VAR
	m_Out:INT;
	m_in: LREAL;
END_VAR

IF Enable THEN
	IF ABS(MaxValue) > 0.0 THEN
		m_in:=LIMIT(0, In, Set_MaxValue);
		m_Out:=REAL_TO_INT(m_In /MaxValue*32767) + AnalogOffset;
		out:=LIMIT(0, m_out, 32767);
	ELSE
		out:=AnalogOffset;
	END_IF
ELSE
	out:=AnalogOffset;
END_IF

END_FUNCTION_BLOCK

// ---- POUs/002_Modbus/PRG_SerialComm.TcPOU
PROGRAM PRG_SerialComm
VAR
	CmdSendData1,CmdSendData2,CmdSendData3		: SendData; //将任何类型的变量的内容发送到与输入变量TxBuffer对应的接口。只要Busy=TRUE，传输就没有完成。当Busy=FALSE和Error=0时，数据已成功发送
	StsReceiveData1,StsReceiveData2	: ReceiveData;
	DataRecive1     :ARRAY[1..16]OF BYTE;	
	Prefix1 : ARRAY[1..5] OF BYTE :=[16#46,16#51,16#0C,16#32,16#02];
	
	Dely1,Dely2:Tc2_Standard.TON;
	clearbuf1,clearbuf2,clearbuf3,clearbuf4:Tc2_SerialCom.ClearComBuffer;
	i,j: INT;
	
	level:ARRAY[1..10] OF LREAL;	
	(*******************UV mode****************************)
	DataSend_uv_mode					:ARRAY[1..11]OF BYTE:=[16#01,16#10,16#00,16#C0,16#00,16#01,16#02,16#00,16#11,16#77,16#5C];//232
	DataRecive_uv_mode	    			:ARRAY[1..8] OF BYTE;
	DataRecive_uv_mode_correct			:ARRAY[1..8] OF BYTE:=[16#01,16#10,16#00,16#C0,16#00,16#01,16#01,16#F5];
	ton_Remote							:Tc2_Standard.TON;
	(*******************UV buad****************************)
	step_burd							:INT;
	DataSend_Buad_set					:ARRAY[1..17] OF BYTE;
	DataSend_Buad						:ARRAY[1..19] OF BYTE;
	DataRecive_Buad_correct				:ARRAY[1..8] OF BYTE:=[16#01,16#10,16#01,16#20,16#00,16#05,16#00,16#3C];
	DataRecive_Buad						:ARRAY[1..8] OF BYTE;
	EN_Buad:DINT;
	HMI_Buad:INT:=2;//1：9600,2:57600,3:115200
	CRC16_Send_Buad:WORD;
	(*******************UV power****************************)
	step_set_power							:INT;
	DataSend_Power_set						:ARRAY[1..41] OF BYTE;
	DataSend_Power						    :ARRAY[1..43] OF BYTE;
	DataReceive_Power						:ARRAY[1..8] OF BYTE;
	CRC16_Send_Power:WORD;
	UV_power_old_L							:DINT;//上一次能量
	UV_power_old_R							:DINT;//上一次能量
	UV_Power_r_trig:						Tc2_Standard.R_TRIG;//能量变化
	UV_Power_send_f_trig					:Tc2_Standard.F_TRIG;
	(*******************UV STATE****************************)
	step_read_state:INT;
	DataSend_State						:ARRAY[1..8] OF BYTE:=[16#01,16#03,16#00,16#CB,16#00,16#1A,16#B5,16#FF];
	DataRecive_State					:ARRAY[1..57] OF BYTE;
	Prefix_DataRecive_State: ARRAY[1..3] OF BYTE :=[16#01,16#03,16#34];
	
	(*******************UV version****************************)
	step_read_version	:INT;
	DataSend_Version	:ARRAY[1..8] OF BYTE:=[16#01,16#03,16#00,16#AE,16#00,16#10,16#25,16#E7];
	DataRecive_Version	:ARRAY[1..37] OF BYTE;
	Prefix_DataRecive_Version: ARRAY[1..3] OF BYTE :=[16#01,16#03,16#20];
	soft_version :ARRAY[0..2] OF WORD;
	soft_date    :ARRAY[0..2] OF WORD;//年，月，日
	hardware_version :ARRAY[0..2] OF WORD;
	hardware_date:ARRAY[0..2] OF WORD;//年，月，日
		
	(*******************UV first light****************************)
	step_first_light        :INT;
	DataSend_First_light	:ARRAY[1..8] OF BYTE:=[16#01,16#03,16#02,16#12,16#00,16#06,16#64,16#75];
	DataRecive_First_light	:ARRAY[1..17] OF BYTE;
	Prefix_DataRecive_First_light: ARRAY[1..3] OF BYTE :=[16#01,16#03,16#0C];
	
	(*******************UV Read the accumulated working time****************************)
	step_acc_working_time       :INT;
	DataSend_Acc_working_time 	:ARRAY[1..8] OF BYTE:=[16#01,16#03,16#00,16#E4,16#00,16#20,16#04,16#25];
	DataRecive_Acc_working_time	:ARRAY[1..69] OF BYTE;
	Prefix_DataRecive_Acc_working_time: ARRAY[1..3] OF BYTE :=[16#01,16#03,16#40];


	
	Receive_data_F_trig:Tc2_Standard.F_TRIG;
	
	TON_Timeout:ARRAY[1..4] OF Tc2_Standard.TON;

	
	Main_step_UV:INT;
	
	
		
	uv_power_left_t,uv_power_right_t:DINT;
	bHibyte,bLobyte:BYTE;
	
	error_count_test:ARRAY[1..10] OF DINT;
	error_trig_test:ARRAY[1..10] OF Tc2_Standard.R_TRIG;
	
	CMD_Burd,CMD_Read_Version,CMD_Read_First_light,CMD_Read_Acc_working_time:BOOL;
	
	ton_case:Tc2_Standard.TON;
	
END_VAR

(****************MainTankLevel***************)
COM1_MainTankLevel();

(*********************************UV**************************************)
(*********************clear buff******************				
Dely1(IN:=NOT Dely1.Q , PT:=T#500MS , Q=> , ET=> );	
IF Dely1.Q THEN 
		clearbuf3(Buffer:=TXBUFFER2  );
		clearbuf4(Buffer:=RXBUFFER2   );	
END_IF
*)
(*****************timeout,自复位***************************)
TON_Timeout[1](IN:= NOT StsReceiveData2.busy  , PT:=T#2S , Q=> , ET=> );
TON_Timeout[2](IN:=StsReceiveData2.busy  , PT:=T#2S , Q=> , ET=> );
IF TON_Timeout[1].Q OR TON_Timeout[2].Q THEN 
	GVL.UV_timeout:=TRUE;
ELSE
	GVL.UV_timeout:=FALSE;
END_IF


(*********************UV_pro*******************)
COM2_UVLed_Set_Power();

IF Axis[1].Ref.Status.NotMoving THEN 
	CASE Main_step_UV OF
	0:
		IF CMD_Burd THEN 
			Main_step_UV:=10;
		ELSIF CMD_Read_Version THEN 
			Main_step_UV:=20;
		ELSIF CMD_Read_First_light THEN 
			Main_step_UV:=30;
		ELSIF CMD_Read_Acc_working_time THEN 
			Main_step_UV:=40;
		ELSE 
			Main_step_UV:=50;
		END_IF
	10://COM2_UVLedburd 
		CMD_Burd:=FALSE;
		_10_COM2_UVLed_burd();
		ton_case(IN:=TRUE , PT:=T#1S , Q=> , ET=> );
		Receive_data_F_trig(CLK:=StsReceiveData2.busy , Q=> );
		IF ton_case.Q OR Receive_data_F_trig.Q  THEN 
			ton_case(IN:=FALSE);
			step_burd:=0;
			Main_step_UV:=0;
		END_IF
	20://CMD_Read_Version
		CMD_Read_Version:=FALSE;
		_20_COM2_UVLed_Version();
		ton_case(IN:=TRUE , PT:=T#1S , Q=> , ET=> );
		Receive_data_F_trig(CLK:=StsReceiveData2.busy , Q=> );
		IF ton_case.Q OR Receive_data_F_trig.Q THEN 
			ton_case(IN:=FALSE);
			step_read_version:=0;
			Main_step_UV:=0;
		END_IF
		
	30://CMD_Read_First_light
		CMD_Read_First_light:=FALSE;
		_30_COM2_UVLed_First_light();
		ton_case(IN:=TRUE , PT:=T#1S , Q=> , ET=> );
		Receive_data_F_trig(CLK:=StsReceiveData2.busy , Q=> );
		IF ton_case.Q THEN 
			ton_case(IN:=FALSE);
			step_first_light:=0;		
			Main_step_UV:=0;
		END_IF
	40://CMD_Read_Acc_working_time
		CMD_Read_Acc_working_time:=FALSE;
		_40_COM2_UVLed_Acc_working_time();
		ton_case(IN:=TRUE , PT:=T#1S , Q=> , ET=> );
		Receive_data_F_trig(CLK:=StsReceiveData2.busy , Q=> );
		IF ton_case.Q THEN 
			ton_case(IN:=FALSE);
			step_acc_working_time:=0;
			Main_step_UV:=0;
		END_IF
	50:		
		_50_COM2_UVLed_Read_State();
		IF CMD_Burd OR CMD_Read_Version OR CMD_Read_First_light OR CMD_Read_Acc_working_time THEN
			Main_step_UV:=0;
		END_IF 
	END_CASE

END_IF

ACTION _10_COM2_UVLed_burd:
IF HMI_Buad=1 THEN  //9600
		DataSend_Buad_set[8]:=16#00;
		DataSend_Buad_set[9]:=16#00;
		DataSend_Buad_set[10]:=16#25;
		DataSend_Buad_set[11]:=16#80;
	ELSIF HMI_Buad=2 THEN //57600
		DataSend_Buad_set[8]:=16#00;
		DataSend_Buad_set[9]:=16#00;
		DataSend_Buad_set[10]:=16#E1;
		DataSend_Buad_set[11]:=16#00;
	ELSIF HMI_Buad=3 THEN //115200
		DataSend_Buad_set[8]:=16#00;
		DataSend_Buad_set[9]:=16#01;
		DataSend_Buad_set[10]:=16#C2;
		DataSend_Buad_set[11]:=16#00;
	END_IF
	DataSend_Buad_set[1]:=16#01; DataSend_Buad_set[2]:=16#10;DataSend_Buad_set[3]:=16#01;
	DataSend_Buad_set[4]:=16#20; DataSend_Buad_set[5]:=16#00;DataSend_Buad_set[6]:=16#05;
	DataSend_Buad_set[7]:=16#0A; 
	DataSend_Buad_set[12]:=16#00; DataSend_Buad_set[13]:=16#00;//校验位
	DataSend_Buad_set[14]:=16#00;DataSend_Buad_set[15]:=16#08;//停止位
	DataSend_Buad_set[16]:=16#00;DataSend_Buad_set[17]:=16#01;//奇偶校验

	MEMCPY(destAddr:=ADR(DataSend_Buad) , srcAddr:=ADR(DataSend_Buad_set) , n:=SIZEOF(DataSend_Buad_set) );
	
	CRC16_Send_Buad:=MEM.CRC16_Modbus(pMemoryBlock:= ADR(DataSend_Buad_set) , uiLength:=SIZEOF(DataSend_Buad_set) );	
	DataSend_Buad[19]:=WORD_TO_BYTE(CRC16_Send_Buad/255);  // crc h
	DataSend_Buad[18]:=WORD_TO_BYTE(CRC16_Send_Buad);			//CRCL
CASE step_burd OF
0://
10://波特率设置	
	IF NOT  StsReceiveData2.busy THEN 
		CmdSendData2(
			pSendData:= ADR(DataSend_Buad), 
			Length:= 19, 
			Busy=> , 
			Error=> , 
			TXbuffer:= TXBUFFER2);
		step_burd:=20;
	END_IF
20://	接收，比较  波特率
		StsReceiveData2(
			pPrefix:= , 
			LenPrefix:=, 
			pSuffix:= , 
			LenSuffix:= , 
			pReceiveData:= ADR(DataRecive_Buad), 
			SizeReceiveData:= SIZEOF(DataRecive_Buad), 
			Timeout:=T#500MS , 
			Reset:= , 
			DataReceived=> , 
			busy=> , 
			Error=> , 
			RxTimeout=> , 
			LenReceiveData=> , 
			RXbuffer:= RXBUFFER2);
			
			EN_Buad:=MEMCMP(pBuf1:=ADR(DataRecive_Buad) , pBuf2:=ADR(DataRecive_Buad_correct) , n:=SIZEOF(DataRecive_Buad_correct) );
			
			//step_burd:=0;

			
END_CASE
(*
40://  接收，比较  模式
 	StsReceiveData2(
		pPrefix:= , 
		LenPrefix:=, 
		pSuffix:= , 
		LenSuffix:= , 
		pReceiveData:= ADR(DataRecive_uv_mode), 
		SizeReceiveData:= SIZEOF(DataRecive_uv_mode), 
		Timeout:=T#500MS , 
		Reset:= , 
		DataReceived=> , 
		busy=> , 
		Error=> , 
		RxTimeout=> , 
		LenReceiveData=> , 
		RXbuffer:= RXBUFFER2);
	
 	EN_mode:=MEMCMP(pBuf1:=ADR(DataRecive_uv_mode) , pBuf2:=ADR(DataRecive_uv_mode_correct) , n:=SIZEOF(DataRecive_uv_mode_correct) );
	step_UV:=0;
	(*IF EN_mode=0 THEN 
		step_UV:=0;
	ELSE 
		step_UV:=200;
	END_IF
	*)
*)
END_ACTION

ACTION _20_COM2_UVLed_Version:
CASE step_read_version OF 		
0:
	CmdSendData2(
				pSendData:= ADR(DataSend_Version), 
				Length:= 8, 
				Busy=> , 
				Error=> , 
				TXbuffer:= TXBUFFER2);
		step_read_version:=10;
10:		
		StsReceiveData2(
				pPrefix:=ADR(Prefix_DataRecive_Version) , 
				LenPrefix:=3, 
				pSuffix:= , 
				LenSuffix:= , 
				pReceiveData:= ADR(DataRecive_Version), 
				SizeReceiveData:= SIZEOF(DataRecive_Version), 
				Timeout:=T#500MS , 
				Reset:= , 
				DataReceived=> , 
				busy=> , 
				Error=> , 
				RxTimeout=> , 
				LenReceiveData=> , 
				RXbuffer:= RXBUFFER2);
		
		
20:
		;
END_CASE
END_ACTION

ACTION _30_COM2_UVLed_First_light:
CASE step_first_light OF 		
0:
	CmdSendData2(
				pSendData:= ADR(DataSend_First_light), 
				Length:= 8, 
				Busy=> , 
				Error=> , 
				TXbuffer:= TXBUFFER2);
		step_read_version:=10;
10:		
		StsReceiveData2(
				pPrefix:=ADR(Prefix_DataRecive_First_light) , 
				LenPrefix:=3, 
				pSuffix:= , 
				LenSuffix:= , 
				pReceiveData:= ADR(DataRecive_First_light), 
				SizeReceiveData:= SIZEOF(DataRecive_First_light), 
				Timeout:=T#500MS , 
				Reset:= , 
				DataReceived=> , 
				busy=> , 
				Error=> , 
				RxTimeout=> , 
				LenReceiveData=> , 
				RXbuffer:= RXBUFFER2);
		
20:
		;
END_CASE
END_ACTION

ACTION _40_COM2_UVLed_Acc_working_time:
CASE step_acc_working_time OF 		
0:
	CmdSendData2(
				pSendData:= ADR(DataSend_Acc_working_time), 
				Length:= 8, 
				Busy=> , 
				Error=> , 
				TXbuffer:= TXBUFFER2);
		step_read_version:=10;
10:		
		StsReceiveData2(
				pPrefix:=ADR(Prefix_DataRecive_Acc_working_time) , 
				LenPrefix:=3, 
				pSuffix:= , 
				LenSuffix:= , 
				pReceiveData:= ADR(DataRecive_Acc_working_time), 
				SizeReceiveData:= SIZEOF(DataRecive_Acc_working_time), 
				Timeout:=T#500MS , 
				Reset:= , 
				DataReceived=> , 
				busy=> , 
				Error=> , 
				RxTimeout=> , 
				LenReceiveData=> , 
				RXbuffer:= RXBUFFER2);
		
20:
		;
END_CASE
END_ACTION

ACTION _50_COM2_UVLed_Read_State:
(**************读取灯的能量和温度**************************************************)
GVL.HMI_TEMP_L:=BYTE_TO_INT(DataRecive_State[7]);
GVL.HMI_TEMP_R:=BYTE_TO_INT(DataRecive_State[11]);
GVL.HMI_power_L:=BYTE_TO_INT(DataRecive_State[5]);
GVL.HMI_power_R:=BYTE_TO_INT(DataRecive_State[9]);

(******************************************main*****************************************
		StsReceiveData2(
				pPrefix:=ADR(Prefix_DataRecive_State) , 
				LenPrefix:=3, 
				pSuffix:= , 
				LenSuffix:= , 
				pReceiveData:= ADR(DataRecive_State), 
				SizeReceiveData:= SIZEOF(DataRecive_State), 
				Timeout:=T#500MS , 
				Reset:= , 
				DataReceived=> , 
				busy=> , 
				Error=> , 
				RxTimeout=> , 
				LenReceiveData=> , 
				RXbuffer:= RXBUFFER2);
		*)
CASE step_read_state  OF
	
0://读状态，发送
	Dely2(IN:=NOT Dely2.Q  , PT:=T#1000MS , Q=> , ET=> );	
	IF Dely2.Q  THEN 
		
		CmdSendData2(
				pSendData:= ADR(DataSend_State), 
				Length:= 8, 
				Busy=> , 
				Error=> , 
				TXbuffer:= TXBUFFER2);
		step_read_state:=10;    
	END_IF     
10://接收
	Dely2(IN:=false);
	StsReceiveData2(
				pPrefix:=ADR(Prefix_DataRecive_State) , 
				LenPrefix:=3, 
				pSuffix:= , 
				LenSuffix:= , 
				pReceiveData:= ADR(DataRecive_State), 
				SizeReceiveData:= SIZEOF(DataRecive_State), 
				Timeout:=T#500MS , 
				Reset:= , 
				DataReceived=> , 
				busy=> , 
				Error=> , 
				RxTimeout=> , 
				LenReceiveData=> , 
				RXbuffer:= RXBUFFER2);
		step_read_state:=20;  
20://处理数据	 	
		IF DataRecive_State[7]=16#FF THEN //温度异常
				GVL.UV_error_L:=TRUE;
				step_read_state:=100;
		ELSIF  DataRecive_State[11]=16#FF THEN //温度异常
				GVL.UV_error_R:=TRUE;
				step_read_state:=100;	
		ELSIF	DataRecive_State[13]<>16#11	THEN 	//不是232控制
				step_read_state:=30;
		ELSIF  	DataRecive_State[13]=16#11 AND DataRecive_State[7]<>16#FF AND 
			DataRecive_State[11]<>16#FF AND NOT  GVL.UV_error_L  AND NOT GVL.UV_error_R THEN 
				step_read_state:=0;		
		END_IF
		//step_read_state:=0;
30://设定模式RS232		
	   CmdSendData2(
			pSendData:= ADR(DataSend_uv_mode), 
			Length:= 11, 
			Busy=> , 
			Error=> , 
			TXbuffer:= TXBUFFER2);	
   		step_read_state:=0;
					
100://error
			IF GVL_API.stUVLed[1].SetOff OR  GVL_API.stUVLed[2].SetOff THEN 
				GVL.UV_error_L:=FALSE;
				GVL.UV_error_R:=FALSE;
				step_read_state:=0;
			END_IF				
END_CASE
(**************remote***********************)
ton_Remote(IN:=DataRecive_State[13]<>16#11 , PT:=T#5S , Q=> , ET=> );
IF DataRecive_State[13]=16#11 THEN 
	GVL.UVisRemote:=TRUE;
ELSIF ton_Remote.Q THEN 
	GVL.UVisRemote:=FALSE;
END_IF
END_ACTION

ACTION COM1_MainTankLevel:
(************************通讯参数设置*******************)
//Dely1(IN:=TRUE , PT:=T#100MS , Q=> , ET=> );

StsReceiveData1(
	pPrefix:=ADR(Prefix1) , 
	LenPrefix:=5 , 
	pSuffix:= , 
	LenSuffix:= , 
	pReceiveData:= ADR(DataRecive1), 
	SizeReceiveData:= SIZEOF(DataRecive1), 
	Timeout:=T#500MS , 
	Reset:= , 
	DataReceived=> , 
	busy=> , 
	Error=> , 
	RxTimeout=> , 
	LenReceiveData=> , 
	RXbuffer:= RXBUFFER1);

(****************计算********************)
FOR i:=6 TO 15 DO 
	IF DataRecive1[i]<>255 AND DataRecive1[i]<=10 THEN 
		level[i-5]:=BYTE_TO_LREAL(DataRecive1[i]);
	ELSE
		level[i-5]:=0;
	END_IF
END_FOR
GVL.MainTankLevel[1]:=level[5];//LC
GVL.MainTankLevel[2]:=level[6];//LM
GVL.MainTankLevel[3]:=level[4];//Y
GVL.MainTankLevel[4]:=level[3];//M
GVL.MainTankLevel[5]:=level[2];//C
GVL.MainTankLevel[6]:=level[1];//K
GVL.MainTankLevel[7]:=level[7];//W
GVL.MainTankLevel[8]:=level[8];//P
GVL.MainTankLevel[9]:=level[9];//FU
GVL.MainTankLevel[10]:=level[10];//WAST

(*****************timeout,自复位***************************)
TON_Timeout[3](IN:= NOT StsReceiveData1.busy  , PT:=T#2S , Q=> , ET=> );
TON_Timeout[4](IN:=StsReceiveData1.busy  , PT:=T#2S , Q=> , ET=> );
IF TON_Timeout[3].Q OR TON_Timeout[4].Q THEN 
	gvl.MainTankLevel_timeout:=TRUE;
ELSE
	gvl.MainTankLevel_timeout:=FALSE;
END_IF
END_ACTION

ACTION COM2_UVLed_1:
GVL.HMI_TEMP_L:=BYTE_TO_INT(DataRecive_State[7]);
GVL.HMI_TEMP_R:=BYTE_TO_INT(DataRecive_State[11]);
GVL.HMI_power_L:=BYTE_TO_INT(DataRecive_State[5]);
GVL.HMI_power_R:=BYTE_TO_INT(DataRecive_State[9]);
(******************************************UV******************************************)
Dely2(IN:=NOT Dely2.Q  , PT:=T#100MS , Q=> , ET=> );	
IF Dely2.Q AND NOT UV_Power_r_trig.Q THEN 
		CmdSendData2(
				pSendData:= ADR(DataSend_State), 
				Length:= 8, 
				Busy=> , 
				Error=> , 
				TXbuffer:= TXBUFFER2);	
		
END_IF
		StsReceiveData2(
				pPrefix:=ADR(Prefix_DataRecive_State) , 
				LenPrefix:=3, 
				pSuffix:= , 
				LenSuffix:= , 
				pReceiveData:= ADR(DataRecive_State), 
				SizeReceiveData:= SIZEOF(DataRecive_State), 
				Timeout:=T#500MS , 
				Reset:= , 
				DataReceived=> , 
				busy=> , 
				Error=> , 
				RxTimeout=> , 
				LenReceiveData=> , 
				RXbuffer:= RXBUFFER2);
				
(******************************************clear buff******************************************)				
Dely1(IN:=NOT Dely1.Q , PT:=T#500MS , Q=> , ET=> );	
IF Dely1.Q THEN 
		clearbuf3(Buffer:=TXBUFFER2  );
		clearbuf4(Buffer:=RXBUFFER2   );	
END_IF

(******************************************main******************************************)
CASE step_read_state  OF		
0://处理数据
		IF DataRecive_State[7]=16#FF THEN //温度异常
				GVL.UV_error_L:=TRUE;
				step_read_state:=50;
		ELSIF  DataRecive_State[11]=16#FF THEN //温度异常
				GVL.UV_error_R:=TRUE;
				step_read_state:=50;	
		ELSIF	DataRecive_State[13]<>16#11	THEN 	//不是232控制
				step_read_state:=30;
		ELSIF  	DataRecive_State[13]=16#11 AND DataRecive_State[7]<>16#FF AND 
			DataRecive_State[11]<>16#FF AND NOT  GVL.UV_error_L  AND NOT GVL.UV_error_R THEN 
				step_read_state:=50;		//状态正常，设置能量
		END_IF

30://设定模式RS232		
	   CmdSendData2(
			pSendData:= ADR(DataSend_uv_mode), 
			Length:= 11, 
			Busy=> , 
			Error=> , 
			TXbuffer:= TXBUFFER2);	
   		step_read_state:=0;


50:	//	设置能量
		IF NOT GVL.UV_error_L AND NOT  GVL.UV_error_R THEN 
			DataSend_Power_set[8]:=16#00;DataSend_Power_set[9]:=16#11;	//命令
		ELSE
			DataSend_Power_set[8]:=16#00;DataSend_Power_set[9]:=16#00;	//命令	停机
		END_IF
		
		DataSend_Power_set[1]:=16#01;DataSend_Power_set[2]:=16#10;
		DataSend_Power_set[3]:=16#01;DataSend_Power_set[4]:=16#A0;
		DataSend_Power_set[5]:=16#00;DataSend_Power_set[6]:=16#11;
		DataSend_Power_set[7]:=16#22;
		
		
		DataSend_Power_set[10]:=16#00;
		DataSend_Power_set[11]:=DINT_TO_BYTE(GVL.set_uv_power_left);//灯0能量100
		///DataSend_Power_set[11]:=DINT_TO_BYTE(uv_power_left_t);//灯0能量100
		DataSend_Power_set[12]:=16#00;DataSend_Power_set[13]:=GVL.set_uv_parts_left;//灯0段数最大6
		
		DataSend_Power_set[14]:=16#00;
		DataSend_Power_set[15]:=DINT_TO_BYTE(GVL.set_uv_power_right);//灯1能量100
		//DataSend_Power_set[15]:=DINT_TO_BYTE(uv_power_right_t);//灯1能量100
		DataSend_Power_set[16]:=16#00;DataSend_Power_set[17]:=GVL.set_uv_parts_right;//灯1段数最大6
		FOR j:=18 TO 41 DO 
			DataSend_Power_set[J]:=16#00;
		END_FOR
		
		MEMCPY(destAddr:=ADR(DataSend_Power) , srcAddr:=ADR(DataSend_Power_set) , n:=SIZEOF(DataSend_Power_set) );
		CRC16_Send_Power:=MEM.CRC16_Modbus(pMemoryBlock:= ADR(DataSend_Power_set) , uiLength:=SIZEOF(DataSend_Power_set) );
		DataSend_Power[43]:=WORD_TO_BYTE(CRC16_Send_Power/256);  // crc h
		DataSend_Power[42]:=WORD_TO_BYTE(CRC16_Send_Power);			//CRCL
		//bHibyte:=MEM.HighByte(wValue:=CRC16_Send_Power );
		//bLobyte:=MEM.LowByte(wValue:=CRC16_Send_Power );
		
	(*****************检测能量设置变化****************************)	
	UV_Power_r_trig(CLK:=UV_power_old_L<>GVL.set_uv_power_left OR UV_power_old_R<> GVL.set_uv_power_right , Q=> );
		//IF GVL.UV_error_L OR   GVL.UV_error_R OR UV_Power_r_trig.Q THEN 
			UV_power_old_L:=GVL.set_uv_power_left;
			UV_power_old_R:=GVL.set_uv_power_right;
			
			
	
		//END_IF
		
		IF NOT GVL.UV_error_L AND NOT  GVL.UV_error_R THEN 
			step_read_state:=0;
		ELSE
			step_read_state:=100;	//命令	停机
		END_IF
							
100://error
			IF GVL_API.stUVLed[1].SetOff OR  GVL_API.stUVLed[2].SetOff THEN 
				GVL.UV_error_L:=FALSE;
				GVL.UV_error_R:=FALSE;
				step_read_state:=0;
			END_IF			
END_CASE

			CmdSendData3(
					pSendData:= ADR(DataSend_Power), 
					Length:= SIZEOF(DataSend_Power), 
					Busy=> , 
					Error=> , 
					TXbuffer:= TXBUFFER2);	


	 
	 
(*****************timeout,自复位***************************)
TON_Timeout[1](IN:= NOT StsReceiveData2.busy  , PT:=T#2S , Q=> , ET=> );
TON_Timeout[2](IN:=StsReceiveData2.busy  , PT:=T#2S , Q=> , ET=> );
IF TON_Timeout[1].Q OR TON_Timeout[2].Q THEN 
	GVL.UV_timeout:=TRUE;
ELSE
	GVL.UV_timeout:=FALSE;
END_IF
END_ACTION

ACTION COM2_UVLed_Set_Power:
//设置能量
		IF NOT GVL.UV_error_L AND NOT  GVL.UV_error_R THEN 
			DataSend_Power_set[8]:=16#00;DataSend_Power_set[9]:=16#11;	//命令
		ELSE
			DataSend_Power_set[8]:=16#00;DataSend_Power_set[9]:=16#00;	//命令	停机
		END_IF
		
		DataSend_Power_set[1]:=16#01;DataSend_Power_set[2]:=16#10;
		DataSend_Power_set[3]:=16#01;DataSend_Power_set[4]:=16#A0;
		DataSend_Power_set[5]:=16#00;DataSend_Power_set[6]:=16#11;
		DataSend_Power_set[7]:=16#22;
		
		
		DataSend_Power_set[10]:=16#00;
		
		DataSend_Power_set[11]:=DINT_TO_BYTE(GVL.set_uv_power_left);//灯0能量100
		//DataSend_Power_set[11]:=DINT_TO_BYTE(uv_power_left_t);//灯0能量100
		
		DataSend_Power_set[12]:=16#00;DataSend_Power_set[13]:=GVL.set_uv_parts_left;//灯0段数最大6
		
		DataSend_Power_set[14]:=16#00;
		
		DataSend_Power_set[15]:=DINT_TO_BYTE(GVL.set_uv_power_right);//灯1能量100
		//DataSend_Power_set[15]:=DINT_TO_BYTE(uv_power_right_t);//灯1能量100
		
		DataSend_Power_set[16]:=16#00;DataSend_Power_set[17]:=GVL.set_uv_parts_right;//灯1段数最大6
		FOR j:=18 TO 41 DO 
			DataSend_Power_set[J]:=16#00;
		END_FOR
		
		MEMCPY(destAddr:=ADR(DataSend_Power) , srcAddr:=ADR(DataSend_Power_set) , n:=SIZEOF(DataSend_Power_set) );
		CRC16_Send_Power:=MEM.CRC16_Modbus(pMemoryBlock:= ADR(DataSend_Power_set) , uiLength:=SIZEOF(DataSend_Power_set) );
		//DataSend_Power[43]:=WORD_TO_BYTE(CRC16_Send_Power/256);  // crc h
		//DataSend_Power[42]:=WORD_TO_BYTE(CRC16_Send_Power);			//CRCL
		DataSend_Power[43]:=MEM.HighByte(wValue:=CRC16_Send_Power);
		DataSend_Power[42]:=MEM.LowByte(wValue:=CRC16_Send_Power);

CmdSendData3(
			pSendData:= ADR(DataSend_Power), 
			Length:= SIZEOF(DataSend_Power), 
			Busy=> , 
			Error=> , 
			TXbuffer:= TXBUFFER2);
	UV_Power_send_f_trig(CLK:=CmdSendData3.Busy , Q=> );
(*
CASE step_set_power OF
0:
(*****************检测能量设置变化****************************)
UV_Power_r_trig(CLK:=UV_power_old_L<>GVL.set_uv_power_left OR UV_power_old_R<> GVL.set_uv_power_right , Q=> );
	IF UV_Power_r_trig.Q THEN 
			UV_power_old_L:=GVL.set_uv_power_left;
			UV_power_old_R:=GVL.set_uv_power_right;
		step_set_power:=10;
	END_IF
10:
	CmdSendData3(
			pSendData:= ADR(DataSend_Power), 
			Length:= SIZEOF(DataSend_Power), 
			Busy=> , 
			Error=> , 
			TXbuffer:= TXBUFFER2);
	UV_Power_send_f_trig(CLK:=CmdSendData3.Busy , Q=> );
	//IF UV_Power_send_f_trig.Q AND CmdSendData3.Error=0 THEN 
			step_set_power:=0;
	//END_IF
END_CASE
*)
END_ACTION

END_PROGRAM

// ---- POUs/002_Modbus/P_Modbus_RTU.TcPOU
PROGRAM P_Modbus_RTU
VAR
	(*********************RTU******************************)
	master:ARRAY[1..2] OF    ModbusRtuMaster_KL6x22B;
    start:ARRAY[1..2] OF  BOOL:=[TRUE];
	step:ARRAY[1..2] OF  INT;
	
	com1_station:ARRAY[1..5] OF stRtu;
	
	tab_vac_measure	:ARRAY[1..2] OF WORD;//负压表值
	tab_vac_set		:ARRAY[1..2] OF WORD;//负压表值
	sub_pressure_measure	: LREAL;//sub测量正压
	sub_pressure_set		: LREAL;//sun正压设定值
	sub_vac_c_measure		: LREAL;//sub彩色负压值
	sub_vac_w_measure		: LREAL;//sub白色负压值
	sub_vac_c_set			: LREAL;//sub彩色负压设定值
	sub_vac_w_set			: LREAL;//sub白色负压设定值
	
	cycle_time:INT;
	count_time:INT:=5;
	i,j:INT;	
	error_trig :ARRAY[1..10] OF Tc2_Standard.R_TRIG;
	error_count:ARRAY[1..10] OF DINT;//错误计数
	station_error_trig:ARRAY[1..10] OF Tc2_Standard.R_TRIG;	
	station_error AT%Q*:ARRAY[1..10] OF BOOL;
	test_send:BOOL;
END_VAR

VAR PERSISTENT
	break_systime:ARRAY[1..10] OF DATE_AND_TIME;
END_VAR

ACT();

(******************************************台面负压****************************************************)
	(*原本接收10代表1KPA，但修改温控表，使10代表1*)
	(**********READ****负数=正数按位取反+1******************************)
	IF com1_station[1]._04readarray[1].15=0 THEN 
		GVL_API.stTableVacuum[1].vacuum_measured:=WORD_TO_LREAL(com1_station[1]._04readarray[1])/100;
	ELSE 
		GVL_API.stTableVacuum[1].vacuum_measured:=WORD_TO_LREAL(NOT(com1_station[1]._04readarray[1]-1))/100;
	END_IF
	(***************台面负压****write****)	
	com1_station[1]._06writesinglearray[1]:=NOT (LREAL_TO_WORD(GVL_API.stTableVacuum[1].setpoint*100))+1;///负数，反吗+1
	(***************台面负压****writPID*)
	IF 	GVL_API.stTableVacuum[1].ctrlP >0 THEN 	//P 不能为0
		com1_station[1]._06writesinglearray_PID[2]:=LREAL_TO_WORD(GVL_API.stTableVacuum[1].ctrlP*10);//制冷端P
	ELSE 
		com1_station[1]._06writesinglearray_PID[2]:=LREAL_TO_WORD(10*10);//制冷端P
	END_IF
		com1_station[1]._06writesinglearray_PID[4]:=LREAL_TO_WORD(GVL_API.stTableVacuum[1].ctrlI);
		com1_station[1]._06writesinglearray_PID[6]:=LREAL_TO_WORD(GVL_API.stTableVacuum[1].ctrlD);
	
		
(***************温湿度****************)
		gvl.humidity_measured:=	WORD_TO_LREAL(com1_station[3]._03readarray[1])/10;
		IF com1_station[3]._03readarray[1].15=0 THEN 
			gvl.temp_measured:=WORD_TO_LREAL(com1_station[3]._03readarray[2])/10;
		ELSIF com1_station[3]._03readarray[1].15=1 THEN
			gvl.temp_measured:= WORD_TO_LREAL(NOT(com1_station[3]._03readarray[2]-1))/10;
		END_IF
		
		
		
(**************二级墨盒正负压****************
	(**********SUB VAC 正压**************)
	sub_pressure_measure:=  WORD_TO_LREAL( com1_station[4]._03readarray[1])/1000;   //当前值
	
	com1_station[4]._03writearray[1]:=LREAL_TO_WORD(sub_pressure_set*1000);//正压设定
	com1_station[4]._03writearray[4]:=1;//正压自启动
	com1_station[4]._03writearray[4]:=12;//正压电机速度
	
	(**********SUB VAC 负压**************)
	sub_vac_c_measure:=WORD_TO_LREAL(com1_station[5]._03readarray[1])/1000;
	sub_vac_w_measure:=WORD_TO_LREAL(com1_station[5]._03readarray[2])/1000;
	
	com1_station[5]._03writearray[1]:=LREAL_TO_WORD(sub_vac_c_set*1000);
	com1_station[5]._03writearray[2]:=LREAL_TO_WORD(sub_vac_w_set*1000);
	com1_station[5]._03writearray[3]:=3;
	com1_station[5]._03writearray[4]:=3;
*)

ACTION ACT:
CASE step[1] OF 
0: //初始状态
		IF start[1] THEN
			step[1]:=10;
			cycle_time:=0;
		END_IF	
10://站1 04口读操作  真空吸附			
			IF cycle_time>=count_time THEN 
				cycle_time:=0;	
				FOR j:=1 TO 10 DO 
					error_count[j]:=0;
				END_FOR		
			END_IF
						
			master[1].ReadInputRegs(
				UnitID:= 1, 
				Quantity:=4, 
				MBAddr:= 16#03E8, 
				cbLength:= SIZEOF(com1_station[1]._04readarray), 
				pMemoryAddr:= ADR(com1_station[1]._04readarray), 
				Execute:= TRUE, 
				Timeout:= T#200MS);	
											
				IF NOT master[1].BUSY  THEN
					master[1].ReadRegs(Execute:= FALSE, );
					cycle_time:=cycle_time+1;
					step[1]:=20;									
				END_IF
				
				station_error_trig[1](CLK:=master[1].error , Q=> );	
				IF station_error_trig[1].Q THEN 
					error_count[1]:=error_count[1]+1;
				END_IF
20://站1 06口写操作	,设定负压	
			master[1].WriteSingleRegister(
				UnitID:= 1, 
				Quantity:=1, 
				MBAddr:= 0, 
				cbLength:= 2, 
				pMemoryAddr:= ADR(com1_station[1]._06writesinglearray[1]), 
				Execute:= TRUE, 
				Timeout:= T#200MS, 
				BUSY=> , 
				Error=> , 
				ErrorId=> , 
				cbRead=> );			
						
				IF NOT master[1].BUSY  THEN
					master[1].ReadRegs(Execute:= FALSE, );
					step[1]:=21;									
				END_IF
				
				station_error_trig[1](CLK:=master[1].error , Q=> );	
				IF station_error_trig[1].Q THEN 
					error_count[1]:=error_count[1]+1;
				END_IF
21://站1 06口写操作	,设定PID
			master[1].WriteRegs(
				UnitID:= 1, 
				Quantity:=SIZEOF(com1_station[1]._06writesinglearray_PID)/2, 
				MBAddr:= 16#0065, 
				cbLength:= SIZEOF(com1_station[1]._06writesinglearray_PID), 
				pMemoryAddr:= ADR(com1_station[1]._06writesinglearray_PID), 
				Execute:= TRUE, 
				Timeout:= T#200MS, 
				BUSY=> , 
				Error=> , 
				ErrorId=> , 
				cbRead=> );	
				
				
				station_error_trig[1](CLK:=master[1].error , Q=> );	
				IF station_error_trig[1].Q THEN 
					error_count[1]:=error_count[1]+1;
				END_IF	
				IF cycle_time=count_time AND error_count[1]>=2 THEN 
					station_error[1]:=TRUE;
				END_IF

				IF NOT master[1].BUSY  THEN
					master[1].ReadRegs(Execute:= FALSE );
					step[1]:=50;											              		
				END_IF	
(*3://站2 04口读操作
			master[1].ReadInputRegs(
				UnitID:= 2, 
				Quantity:=4, 
				MBAddr:= 16#03E8, 
				cbLength:= SIZEOF(com1_station[2]._04readarray), 
				pMemoryAddr:= ADR(com1_station[2]._04readarray), 
				Execute:= TRUE, 
				Timeout:= T#200MS, 
				 );	
					          
				station_error_trig[2](CLK:=master[1].error , Q=> );	
				IF station_error_trig[2].Q THEN 
					error_count_test[2]:=error_count_test[2]+1;
				END_IF	 
				IF cycle_time=count_time AND error_count_test[2]>=2 THEN 
					station_error[2]:=TRUE;
				END_IF

	
				IF NOT master[1].BUSY  THEN
					master[1].ReadRegs(Execute:= FALSE, );
					IF NOT station_error[2] THEN 
						step[1]:=4;									
					ELSIF station_error[2] THEN 
						step[1]:=5;	
					END_IF		              		
				END_IF					 	
4://站2 06口写操作			
			master[1].WriteSingleRegister(
				UnitID:= 2, 
				Quantity:=1, 
				MBAddr:= 0, 
				cbLength:= SIZEOF(com1_station[2]._06writesinglearray[1]), 
				pMemoryAddr:= ADR(com1_station[2]._06writesinglearray[1]), 
				Execute:= TRUE, 
				Timeout:= T#200MS, 
				BUSY=> , 
				Error=> , 
				ErrorId=> , 
				cbRead=> );			
				
			
				station_error_trig[2](CLK:=master[1].error , Q=> );	
				IF station_error_trig[2].Q THEN 
					error_count_test[2]:=error_count_test[2]+1;
				END_IF	
				IF cycle_time=count_time AND error_count_test[2]>=2 THEN 
					station_error[2]:=TRUE;
				END_IF

				IF NOT master[1].BUSY  THEN
					master[1].ReadRegs(Execute:= FALSE, );					
					IF NOT station_error[2] THEN 
						step[1]:=5;									
					ELSIF station_error[2] THEN 
						step[1]:=5;	
					END_IF		              		
				END_IF		
*)				 	
50://站3温湿度 03读
			master[1].ReadRegs(
				UnitID:= 3, 
				Quantity:=2, 
				MBAddr:= 0, 
				cbLength:= SIZEOF(com1_station[3]._03readarray), 
				pMemoryAddr:= ADR(com1_station[3]._03readarray), 
				Execute:= TRUE, 
				Timeout:= T#200MS, 
				 );	
							     
				station_error_trig[3](CLK:=master[1].error , Q=> );	
				IF station_error_trig[3].Q THEN 
					error_count[3]:=error_count[3]+1;
				END_IF
				IF cycle_time=count_time AND error_count[3]>=2 THEN 
					station_error[3]:=TRUE;
				END_IF
								
				IF NOT master[1].BUSY  THEN
					master[1].ReadRegs(Execute:= FALSE, );										
					step[1]:=10;															              		
				END_IF
				
(*							
6://站4，正压板 03口读操作  当前压墨板正压传感器值，单位0.1kPa	
	     master[1].ReadRegs(
				UnitID:= 16#48, 
				Quantity:=7, 
				MBAddr:= 0, 
				cbLength:= SIZEOF(com1_station[4]._03readarray), 
				pMemoryAddr:= ADR(com1_station[4]._03readarray), 
				Execute:= TRUE, 
				Timeout:= T#200MS, 
				 );	
							
				station_error_trig[4](CLK:=master[1].error , Q=> );	
				IF station_error_trig[4].Q THEN 
					error_count_test[4]:=error_count_test[4]+1;
				END_IF		
			
				IF cycle_time=count_time AND error_count_test[4]>=2 THEN 
					station_error[4]:=TRUE;
				END_IF
				
				IF NOT master[1].BUSY  THEN
					master[1].ReadRegs(Execute:= FALSE, );					
					IF NOT station_error[4] THEN 
						step[1]:=7;									
					ELSIF station_error[4] THEN 
						step[1]:=8;	
					END_IF		              		
				END_IF						     					
7://站4，正压板 03口写操作 设定的压墨值，单位0.1kPa，绝对值。
		master[1].WriteRegs(
				UnitID:= 16#48, 
				Quantity:=6, 
				MBAddr:= 1, 
				cbLength:= SIZEOF(com1_station[4]._03writearray), 
				pMemoryAddr:= ADR(com1_station[4]._03writearray), 
				Execute:= TRUE, 
				Timeout:= T#200MS, 
				BUSY=> , 
				Error=> , 
				ErrorId=> , 
				cbRead=> );			
						
				station_error_trig[4](CLK:=master[1].error , Q=> );	
				IF station_error_trig[4].Q THEN 
					error_count_test[4]:=error_count_test[4]+1;
				END_IF	
				IF cycle_time=count_time AND error_count_test[4]>=2 THEN 
					station_error[4]:=TRUE;
				END_IF
				
				IF NOT master[1].BUSY  AND NOT station_error[4]THEN
					master[1].ReadRegs(Execute:= FALSE, );	
					step[1]:=8;
				ELSIF station_error[4] THEN 
					step[1]:=8;
				END_IF
				IF NOT master[1].BUSY  THEN
					master[1].ReadRegs(Execute:= FALSE, );					
					IF NOT station_error[4] THEN 
						step[1]:=8;									
					ELSIF station_error[4] THEN 
						step[1]:=8;	
					END_IF		              		
				END_IF					     				
8://zhan 5负压板 03口读操作
		master[1].ReadRegs(
				UnitID:= 16#1D, 
				Quantity:=8, 
				MBAddr:= 0, 
				cbLength:= SIZEOF(com1_station[5]._03readarray), 
				pMemoryAddr:= ADR(com1_station[5]._03readarray), 
				Execute:= TRUE, 
				Timeout:= T#200MS, 
				 );	
				
				station_error_trig[5](CLK:=master[1].error , Q=> );	
				IF station_error_trig[5].Q THEN 
					error_count_test[5]:=error_count_test[5]+1;
				END_IF	

				IF cycle_time=count_time AND error_count_test[5]>=2 THEN 
					station_error[5]:=TRUE;
				END_IF
				
				IF NOT master[1].BUSY  THEN
					master[1].ReadRegs(Execute:= FALSE, );					
					IF NOT station_error[5] THEN 
						step[1]:=9;									
					ELSIF station_error[5] THEN 
						step[1]:=1;	
					END_IF		              		
				END_IF							     
9://zhan 5,负压板 03口写	
		master[1].WriteRegs(
				UnitID:= 16#1D, 
				Quantity:=4, 
				MBAddr:= 2, 
				cbLength:= SIZEOF(com1_station[5]._03writearray), 
				pMemoryAddr:= ADR(com1_station[5]._03writearray), 
				Execute:= TRUE, 
				Timeout:= T#200MS, 
				BUSY=> , 
				Error=> , 
				ErrorId=> , 
				cbRead=> );			
				
		
				station_error_trig[5](CLK:=master[1].error , Q=> );	
				IF station_error_trig[5].Q THEN 
					error_count_test[5]:=error_count_test[5]+1;
				END_IF	
				
				IF cycle_time=count_time AND error_count_test[5]>=2 THEN 
					station_error[5]:=TRUE;
				END_IF
					
				IF NOT master[1].BUSY  THEN
					master[1].ReadRegs(Execute:= FALSE, );					
					IF NOT station_error[5] THEN 
						step[1]:=1;									
					ELSIF station_error[5] THEN 
						step[1]:=1;	
					END_IF		              		
				END_IF	
*)
END_CASE

IF GVL_API.stTableVacuum[1].Setoff (*OR GVL_API.stTableVacuum[2].Setoff*) THEN 
	station_error[1]:=FALSE;
	//station_error[2]:=FALSE;
END_IF
IF   GVL_API.stSystemEnvironment.Reset THEN 
	station_error[3]:=FALSE;
END_IF


FOR i:=1 TO 5 DO
 error_trig[i](CLK:=station_error[i] , Q=> );
	IF  error_trig[i].Q THEN 
		break_systime[i]:=systime.dttime;		
	END_IF
END_FOR
END_ACTION

END_PROGRAM

// ---- POUs/003_Input_Output/P_API_IO.TcPOU
PROGRAM P_API_IO
VAR
END_VAR

gvl_api.stAxis[FastScan].Origin:=Axis[FastScan].IO.snHome;
gvl_api.stAxis[FastScan].LimitP:=Axis[FastScan].IO.snLimitP;
gvl_api.stAxis[Z_Axis].Origin:=Axis[Z_Axis].IO.snHome;
gvl_api.stAxis[Z_Axis].LimitP:=Axis[Z_Axis].IO.snLimitP;

END_PROGRAM

// ---- POUs/010_Motion/MotionBase/FB_Home_Z.TcPOU
FUNCTION_BLOCK FB_Home_Z
(*========================================
Execute需一直有效，功能块才会一直执行
先回原点，然后直接到等待位
==========================================*)
VAR_IN_OUT
	Axis				:AXIS_REF;	(* B *)
END_VAR
VAR_INPUT
	Execute				:BOOL;	(* B *)
	PosLimit			:BOOL;			(*正极限位信号*)
	NegLimit			:BOOL;			(*负极限位信号*)
	Position			:LREAL			(* B *) := DEFAULT_HOME_POSITION;
	HomeingVelo			:LREAL:=5;
	Standby_position	:LREAL;		//最终待机位
	bCalibrationCam 	:BOOL;	(* V *)	(* Beckhoff proprietary input *)
	rel_dis         	:LREAL:=10;  //碰到原点后，正向移动距离，在开始寻原点
	TimeOutSet       	:LREAL;//s
	reset				:BOOL;
	maxDistance:LREAL;
END_VAR
VAR_OUTPUT
	Done				:BOOL;	(* B *)
	Busy				:BOOL;	(* E *)
	Active				:BOOL;	(* E *)
	CommandAborted		:BOOL;	(* E *)
	Error				:BOOL;	(* B *)
	ErrorID				:UDINT;	(* E *)
	TimeOut				:BOOL;//回零超时
	HomeErr				:BOOL;//超过最大行程

END_VAR
VAR
	mcJog			:MC_Jog;
	mcHome			:MC_Home;
	mcRel           :MC_MoveRelative;
	mcAbs           :MC_MoveAbsolute;	
	mcStop			:MC_Stop;
	HomeStep		:INT;
	ton				:TON;
	StopDo			:BOOL;
	start_pos		:LREAL;
	start_r_trig:Tc2_Standard.R_TRIG;
END_VAR

ton(IN:=Execute , PT:=LREAL_TO_TIME(TimeOutSet*1000) , Q=> , ET=> );
IF ton.Q THEN 
	TimeOut:=TRUE;
	HomeStep	:=100;
END_IF

start_r_trig(CLK:=Execute , Q=> );
IF start_r_trig.Q THEN 
	start_pos:=Axis.NcToPlc.ActPos;
END_IF


IF  NOT Execute THEN
	mcJog.JogForward		:=FALSE;
	mcJog.JogBackwards		:=FALSE;
	mcHome.Execute			:=FALSE;
	mcRel.Execute			:=FALSE;
	mcAbs.Execute			:=FALSE;
	done					:=FALSE;
	busy					:=FALSE;	
	HomeStep				:=0;
END_IF

IF reset THEN 
	Error					:=FALSE;
	TimeOut					:=FALSE;
	HomeErr			:=FALSE;
END_IF

CASE HomeStep OF

0:
	busy	:=FALSE;
	Done	:=FALSE;
	IF 	Execute AND NOT Error  THEN		
		IF  NOT bCalibrationCam THEN
			HomeStep	:=10;
		ELSE
			HomeStep	:=20;
		END_IF
		busy	:=TRUE;
		ErrorID	:=0;		
	END_IF
	
10:(*先向负限位方向运动*)
	mcJog.JogForward		:=FALSE;
	mcJog.JogBackwards		:=TRUE;		 
	IF	bCalibrationCam THEN
		mcJog.JogBackwards	:=FALSE;		
		HomeStep	:=20;		
	ELSIF mcJog.Error   THEN
			HomeStep	:=100;
	ELSIF ABS(start_pos-Axis.NcToPlc.ActPos)>maxDistance THEN 
			HomeStep	:=100;
			HomeErr:=TRUE;
	END_IF
	
20:(*从原点处正方向移动一段距离*)
	mcRel.Execute		:=TRUE;	
	IF mcRel.Done AND Axis.Status.NotMoving THEN 
		mcRel.Execute	:=FALSE;
		HomeStep		:=30;
	ELSIF mcRel.Error OR TimeOut THEN 
		HomeStep	:=100;	
	END_IF
	
30:(*调用回零功能块*)
	mcHome.Execute	:=TRUE;
	IF mcHome.Done AND AXIS.Status.Homed THEN
		mcHome.Execute	:=FALSE;		
		HomeStep		:=50;
	ELSIF AXIS.Status.Error OR TimeOut THEN
		HomeStep		:=100;
	END_IF
(*	
40:(*碰正极限*)
	mcJog.JogBackwards		:=FALSE;
	mcJog.JogForward		:=TRUE;		(*向正限位方向运动*)	
	IF PosLimit THEN 
		mcJog.JogForward	:=FALSE;
		IF Axis.Status.NotMoving THEN
			HomeStep	:=50;
		END_IF
	ELSIF mcJog.Error OR TimeOut THEN
			HomeStep	:=100; 
	END_IF
*)	
50:(*回待机位*)
	mcAbs.Execute:=TRUE;
	IF mcAbs.Done AND Axis.Status.NotMoving THEN 
		mcAbs.Execute	:=FALSE;
		done			:=TRUE;
		HomeStep		:=99; 		
	END_IF
99:
	;	

100:
	Error			:=TRUE;
	IF	mcHome.ErrorID <> 0 THEN
		ErrorID			:=mcHome.ErrorID;
	ELSIF  mcJog.ErrorID <> 0 THEN
		ErrorID			:=mcJog.ErrorID;
	ELSIF mcRel.ErrorID<>0 THEN 
		ErrorID			:=mcRel.ErrorID;
	ELSIF mcAbs.ErrorID<>0 THEN 
		ErrorID			:=mcAbs.ErrorID;	
	END_IF
	mcJog.JogForward		:=FALSE;
	mcJog.JogBackwards		:=FALSE;
	mcHome.Execute			:=FALSE;
	mcRel.Execute			:=FALSE;
	mcAbs.Execute			:=FALSE;
	StopDo			:=TRUE;
	HomeStep		:=0;
	
END_CASE


Call_FB();

ACTION Call_FB:
Axis.ReadStatus();
mcJog
	(
	Velocity:=	HomeingVelo ,
	Mode:=		MC_JOGMODE_CONTINOUS ,
	Axis:=		Axis ,
	);

mcHome
	(
	Execute:= ,
	Position:=			Position ,
	HomingMode:= 		,
	BufferMode:= 		,
	Options:=			 ,
	bCalibrationCam:=	bCalibrationCam ,
	Axis:=				Axis ,
	);

mcRel(
	Axis:=Axis , 
	Execute:= , 
	Distance:=rel_dis , 
	Velocity:= HomeingVelo, 
	Acceleration:= , 
	Deceleration:= , 
	Jerk:= , 
	BufferMode:= , 
	Options:= , 
	Done=> , 
	Busy=> , 
	Active=> , 
	CommandAborted=> , 
	Error=> , 
	ErrorID=> );
mcAbs(
	Axis:=Axis , 
	Execute:= , 
	Position:=Standby_position , 
	Velocity:=HomeingVelo , 
	Acceleration:= , 
	Deceleration:= , 
	Jerk:= , 
	BufferMode:= , 
	Options:= , 
	Done=> , 
	Busy=> , 
	Active=> , 
	CommandAborted=> , 
	Error=> , 
	ErrorID=> );
mcStop(
	Axis:=Axis , 
	Execute:=StopDo , 
	Deceleration:= , 
	Jerk:= , 
	Options:= , 
	Done=> , 
	Busy=> , 
	Active=> , 
	CommandAborted=> , 
	Error=> , 
	ErrorID=> );
IF mcStop.Busy THEN 
	StopDo:=FALSE;
END_IF
END_ACTION

END_FUNCTION_BLOCK

// ---- POUs/030_MediaTransport/TableVacuum/FB/FB_TableVacuum.TcPOU
FUNCTION_BLOCK FB_TableVacuum
VAR_INPUT
	vacuum_measured			:LREAL;//	Pa
	vacuum_min				:LREAL:=3.5;	//	Pa 3.5
	vacuum_max				:LREAL:=10;	//	Pa	10
	setpoint				:LREAL:=6;	//	Pa	6[0-8]
	vacuum_offset_collector	:LREAL;	//	Pa	Offset used to calibrate the vacuum sensor of the vacuum collector
	setpoint_range_pct		:LREAL:=70;	//	%  Threshold used to indicate the table vacuum is ready
	vacuum_timeout			:LREAL:=6000;	//ms	TIME needed TO reach the vacuum setpoint.
	vacuum_off_timeout		:LREAL:=3000;	//	ms 	Time to turn off the vacuum
	IO_Error				:BOOL;
END_VAR
VAR_OUTPUT
	state					:INT;
	error_code					:INT;
	Run						:BOOL;
	error					:BOOL;
END_VAR
VAR
	step					:INT;
	setpoint_act			:LREAL;
	reach_setpoint_ton		:ton;
	turn_off_ton			:TON;
	turn_on_delay           :Tc2_Standard.TON;
	temp_setpoint			:LREAL;
END_VAR
VAR_IN_OUT
	Initialize				:BOOL;
	SetVacuumOn				:BOOL;
	SetVacuumOff			:BOOL;
	Setoff					:BOOL;
END_VAR


CASE step OF 
0://waiting
	IF Initialize THEN 
		step:=5;
	ELSIF SetVacuumOn THEN 
		step:=10;
	ELSIF SetVacuumOff THEN 
		step:=30;
	ELSIF Setoff OR GVL.Reset THEN 
		step:=50;
	END_IF	
5://off
	Run:=FALSE;
	setpoint_act:=0;
	SetVacuumOn:=FALSE;
	SetVacuumOff:=FALSE;
	Setoff:=FALSE;
	
	
	state:=TabVacStateEnum.off;
	error_code:=TabVacErrorEnum.no_error;
	
	IF Initialize AND 
		setpoint_range_pct<>0 AND vacuum_min>=0 AND vacuum_max>0 THEN 
		Initialize:=FALSE;
		state:=TabVacStateEnum.idle;	
		step:=0;
	END_IF
	
10://INI
	SetVacuumOff:=FALSE;			
	IF setpoint>=vacuum_min AND setpoint<=vacuum_max AND vacuum_timeout>0  THEN 
		setpoint_act:=setpoint;
	ELSIF  setpoint>=vacuum_max THEN 
			setpoint_act:=vacuum_max;
	ELSIF setpoint<=vacuum_min THEN 
		setpoint_act:=vacuum_min;
	END_IF

	IF SetVacuumOn THEN 
			step:=20;
	ELSIF Setoff THEN 
			step:=50;
	END_IF

20://waiting_vacuum_on
	SetVacuumOn:=FALSE;
	Initialize:=FALSE;
	SetVacuumOff:=FALSE;
	
	state:=TabVacStateEnum.waiting_vacuum_on;
	Run:=TRUE;
	reach_setpoint_ton(IN:=TRUE , PT:=LREAL_TO_TIME(vacuum_timeout) , Q=> , ET=> );
	IF reach_setpoint_ton.Q (*AND vacuum_measured/setpoint_act*100<setpoint_range_pct *)THEN		
		error_code:=TabVacErrorEnum.vacuum_on_timeout;
		step:=100;
	END_IF
	(*************转on 用时间******************************)
	(*IF NOT reach_setpoint_ton.Q AND  vacuum_measured/setpoint_act*100>=setpoint_range_pct THEN 	
		reach_setpoint_ton(IN:=FALSE); 		
		state:=TabVacStateEnum.on;	
		step:=0;
	END_IF*)
	
	turn_on_delay(IN:=TRUE , PT:=INT_TO_TIME(HMI_Vac_dely_on), Q=> , ET=> );
	IF NOT reach_setpoint_ton.Q AND  turn_on_delay.Q THEN 	
		reach_setpoint_ton(IN:=FALSE); 	
		turn_on_delay(IN:=FALSE);	
		state:=TabVacStateEnum.on;	
		step:=0;
	END_IF
	
	IF Setoff THEN 
		step:=50;
	END_IF
	
30://on		
	IF SetVacuumOff AND vacuum_off_timeout>0 THEN 
		step:=40;
	ELSIF Setoff THEN 
		step:=50;	
	END_IF
40://waiting_vacuum_off
	Initialize:=FALSE;
	SetVacuumOn:=FALSE;
	Setoff:=FALSE;
	
	SetVacuumOff:=FALSE;
	state:=TabVacStateEnum.waiting_vacuum_off;
	Run:=FALSE;
	turn_off_ton(IN:=TRUE , PT:=LREAL_TO_TIME(vacuum_off_timeout) , Q=> , ET=> );	 
	IF vacuum_measured<setpoint*0.5 AND NOT turn_off_ton.Q  THEN 
		turn_off_ton(IN:=FALSE);
		state:=TabVacStateEnum.idle;
		step:=0;
	ELSIF vacuum_measured>=0 AND turn_off_ton.Q THEN 
		error_code:=TabVacErrorEnum.vacuum_off_timeout;
		step:=100;
	END_IF
50://waiting_off
	Initialize:=FALSE;
	SetVacuumOn:=FALSE;
	SetVacuumOff:=FALSE;

	Setoff:=FALSE;
	state:=TabVacStateEnum.waiting_off;
	error_code:=TabVacErrorEnum.no_error;
	Run:=FALSE;
	error:=FALSE;
	
	IF vacuum_measured<=0.5 THEN 
		state:=TabVacStateEnum.off;
		step:=0;
	END_IF
100://error
	Initialize:=FALSE;
	SetVacuumOn:=FALSE;
	SetVacuumOff:=FALSE;
	
	error:=TRUE;
	state:=TabVacStateEnum.error;
	Run:=FALSE;
	reach_setpoint_ton(IN:=FALSE);
	turn_off_ton(IN:=FALSE);
	step:=0;	
END_CASE

IF Setoff OR GVL.Reset THEN 
	step:=50;
END_IF	
	
IF state<>TabVacStateEnum.off AND state<>TabVacStateEnum.waiting_off AND state<>TabVacStateEnum.error THEN 
	IF IO_Error THEN 
		error_code:=TabVacErrorEnum.unknown_error;
		step:=100;
	END_IF
	IF GVL.Emstop_Button THEN 
		error_code:=TabVacErrorEnum.emergency_error;	
		step:=100;
	END_IF
END_IF

END_FUNCTION_BLOCK

// ---- POUs/040_System/SafetyGuard/FB/FB_SafetyGuard.TcPOU
FUNCTION_BLOCK FB_SafetyGuard
VAR_INPUT
	shuttle_crash_detector						:BOOL;
	emergency_stop									:BOOL;
	limit_switch										:BOOL;
	interlock_triggered								:BOOL;//安全门被触发
	LightCurtainTriggered							:BOOL;
END_VAR
VAR_OUTPUT
	error_code			:INT;
	state						:INT;
	Init_Done				:BOOL;
	Error						:BOOL;
END_VAR
VAR
	step    				:INT;
	ton1					:Tc2_Standard.TON;
END_VAR
VAR_IN_OUT
	Initialize			:BOOL;
	SetOff			:BOOL;
END_VAR

CASE  step OF
0://waiting
	IF Initialize THEN 
		step:=5;
	ELSIF SetOff OR GVL.Reset THEN 
		step:=99;
	END_IF
	
	(******************状态自复位***************************)
	ton1(IN:=Init_Done  , PT:=T#1S , Q=> , ET=> );
	IF ton1.Q THEN 
		Init_Done:=FALSE;
	END_IF
5://OFF
	state:=SafetyGuardStateEnum.off;
	error_code:=SafetyGuardErrorEnum.no_error;
	
	IF Initialize THEN 
		Initialize:=FALSE;
		step:=10;
	END_IF
10://Initializing
	state:=SafetyGuardStateEnum.initializing;
	
	step:=20;
20://ready
	Init_Done:=TRUE;
	state:=SafetyGuardStateEnum.ready;
	step:=0;

99://SetOff
	SetOff:=FALSE;
	Error:=FALSE;
	state:=SafetyGuardStateEnum.off;
	error_code:=SafetyGuardErrorEnum.no_error;
	step:=0;
100://error
		state:=SafetyGuardStateEnum.error;
		Error:=TRUE;
		step:=0;
END_CASE

IF SetOff OR GVL.Reset THEN 
		step:=99;
END_IF

IF state <>SafetyGuardStateEnum.off AND state <>SafetyGuardStateEnum.error THEN 
		IF emergency_stop THEN 
		error_code:=SafetyGuardErrorEnum.emergency_error;
		step:=100;
	ELSIF 	interlock_triggered THEN 
		error_code:=SafetyGuardErrorEnum.interlock_error;
		step:=100;
	ELSIF	shuttle_crash_detector THEN 
		error_code:=SafetyGuardErrorEnum.shuttle_crash_error;
		step:=100;
	ELSIF	limit_switch THEN 
		error_code:=SafetyGuardErrorEnum.limit_switch_error;
		step:=100;
	END_IF
END_IF

END_FUNCTION_BLOCK

// ---- POUs/040_System/SafetyGuard/P_SafetyGuard.TcPOU
PROGRAM P_SafetyGuard
VAR
	i,j:INT;
	FB_SafetyGuard:FB_SafetyGuard;
	log_ErrorEnum:SafetyGuardErrorEnum;
	log_ID:INT;
	trig1,trig2:Tc2_Standard.R_TRIG;
END_VAR

ACT_LOG();
(************************PLC使用****************************************)
		(************Emstop******************)
	//GVL.Emstop:=gvl.HMI_btEmstop;				//	测试用	
	GVL.Emstop_SAFE:=P_TwinSAFE.Emergency_stop_2904 ;
	GVL.Emstop_Button:=P_TwinSAFE.btEmergency_stop;
	GVL.Reset	 :=stInput.btReset;
	
		(************interlock******************)
	FOR i:=1 TO 8 DO 
		IF NOT P_TwinSAFE.biinterlock[i] THEN 
			GVL.interlock_triggered:=TRUE;
			EXIT;
		ELSE 
			GVL.interlock_triggered:=FALSE;			
		END_IF
	END_FOR
	
		(************shuttle_crash******************)
	gvl.shuttle_crash:=NOT P_TwinSAFE.bishuttle_crash_detector_left OR NOT P_TwinSAFE.bishuttle_crash_detector_right;

(************************C#使用****************************************)
	(********左右防撞触发保存******************)
	trig1(CLK:=NOT P_TwinSAFE.bishuttle_crash_detector_left , Q=> );
	IF trig1.Q THEN 
		GVL_API.stSafetyGuard.shuttle_crash_detector_left:=TRUE;
	END_IF
	
	trig1(CLK:=NOT P_TwinSAFE.bishuttle_crash_detector_right , Q=> );
	IF trig1.Q THEN 
		GVL_API.stSafetyGuard.shuttle_crash_detector_right:=TRUE;
	END_IF
	
	IF GVL_API.stSafetyGuard.SetOff THEN 
		GVL_API.stSafetyGuard.shuttle_crash_detector_left:=FALSE;
		GVL_API.stSafetyGuard.shuttle_crash_detector_right:=FALSE;
	END_IF
	
	GVL_API.stSafetyGuard.emergency_stop						:=GVL.Emstop_SAFE;
	GVL_API.stSafetyGuard.shuttle_crash_detector_left			:=NOT P_TwinSAFE.bishuttle_crash_detector_left;
	GVL_API.stSafetyGuard.shuttle_crash_detector_right			:=NOT P_TwinSAFE.bishuttle_crash_detector_right;
	GVL_API.stSafetyGuard.limit_switch_left						:=Axis[FastScan].IO.snLimitN;
	GVL_API.stSafetyGuard.limit_switch_right					:=Axis[FastScan].IO.snLimitP;
	GVL_API.stSafetyGuard.limit_switch_bottom					:=Axis[Z_Axis].IO.snLimitP;
	GVL_API.stSafetyGuard.interlock_front_left					:=NOT P_TwinSAFE.biinterlock[1];
	GVL_API.stSafetyGuard.interlock_front_right					:=NOT P_TwinSAFE.biinterlock[2];
	GVL_API.stSafetyGuard.interlock_rear_left					:=NOT P_TwinSAFE.biinterlock[3];
	GVL_API.stSafetyGuard.interlock_rear_right					:=NOT P_TwinSAFE.biinterlock[4];
	GVL_API.stSafetyGuard.interlock_shuttle_door				:=NOT P_TwinSAFE.biinterlock[5];
	GVL_API.stSafetyGuard.Interlock_maintenace_door				:=NOT P_TwinSAFE.biinterlock[6];
	GVL_API.stSafetyGuard.Interlock_spit_door					:=NOT P_TwinSAFE.biinterlock[7] AND NOT P_TwinSAFE.biinterlock[8];

(**************************FB调用***************************************************)
FB_SafetyGuard(
	shuttle_crash_detector:=gvl.shuttle_crash, 
	emergency_stop:=GVL_API.stSafetyGuard.emergency_stop, 
	limit_switch:= GVL_API.stSafetyGuard.limit_switch_left OR GVL_API.stSafetyGuard.limit_switch_right OR  GVL_API.stSafetyGuard.limit_switch_bottom, 
	interlock_triggered:= gvl.interlock_triggered , 
	LightCurtainTriggered:= , 
	error_code=> GVL_API.stSafetyGuard.error_code, 
	state=> GVL_API.stSafetyGuard.state, 
	Init_Done=>GVL_API.stSafetyGuard.Init_Done , 
	Error=> GVL_API.stSafetyGuard.Error, 
	Initialize:=GVL_API.stSafetyGuard.Initialize , 
	SetOff:=GVL_API.stSafetyGuard.SetOff );

ACTION ACT_LOG:
(*************************LOG*******************************************)
//只记录错误
log_ID:=430;

//ERROR,log_ErrorEnum只能等于一个常数,   
CASE GVL_API.stSafetyGuard.error_code  OF
0	:	log_ErrorEnum	:=	0	;
1	:	log_ErrorEnum	:=	1	;
2	:	log_ErrorEnum	:=	2	;
4	:	log_ErrorEnum	:=	4	;
8	:	log_ErrorEnum	:=	8	;
16	:	log_ErrorEnum	:=	16	;
32	:	log_ErrorEnum	:=	32	;
64	:	log_ErrorEnum	:=	64	;
128	:	log_ErrorEnum	:=	128	;

END_CASE

AlarmActionArray[log_ID+1].AlarmMsg.EN	:=CONCAT('SafetyGuard Error: ',TO_STRING(log_ErrorEnum));
fbSetAlarm[log_ID+1](
	InUse:=TRUE , 
	EventId:=log_ID+1 , 
	EventActive:=GVL_API.stSafetyGuard.error_code<>0 , 
	EventClass:=Alm_EventClass.Alarm , 
	ToTheLogFile:=TRUE, 
	ToTheHistory:=TRUE , 
 );
 
//reset
AlarmActionArray[log_ID+2].AlarmMsg.EN	:=	'SafetyGuard Reset ';
fbSetAlarm[log_ID+2](
	InUse:=TRUE , 
	EventId:=log_ID+2 , 
	EventActive:=GVL_API.stSafetyGuard.SetOff  , 
	EventClass:=Alm_EventClass.Event , 
	ToTheLogFile:=TRUE, 
	ToTheHistory:=TRUE , 
 );
END_ACTION

END_PROGRAM

// ---- POUs/050_InkSystem/P_InkSystem.TcPOU
PROGRAM P_InkSystem
VAR

END_VAR

P_ISS();
P_Stirrer_WastePump();

END_PROGRAM

// ---- POUs/050_InkSystem/搅拌_吸废墨/P_Stirrer_WastePump.TcPOU
PROGRAM P_Stirrer_WastePump
VAR
	(*********搅拌**************)
	FB_Stirrer:FB_Stirrer;	
	EnStirrer: BOOL:=TRUE;
	(*********吸废墨**************)
	FB_waste_pump :FB_Stirrer;
	
END_VAR

FB_Stirrer(
	enable:=HMI_SetStirrer_intervalTime>0 AND HMI_SetStirrer_continueTime>0 AND NOT GVL.Emstop_Button , 
	continueTime:=HMI_SetStirrer_continueTime , 
	intervalTime:=HMI_SetStirrer_intervalTime , 
	PumpWorkingF=>stOutput.bqStirrerWorkingF , 
	PumpWorkingB=>stOutput.bqStirrerWorkingB );
	
FB_waste_pump(
	enable:=NOT GVL.Emstop_Button , 
	continueTime:=HMI_SetWaste_continueTime , 
	intervalTime:=HMI_SetWaste_intervalTime , 
	PumpWorkingF=> , 
	PumpWorkingB=>);
IF FB_waste_pump.PumpWorkingB OR FB_waste_pump.PumpWorkingF THEN 
	stOutput.bqWastePump:=TRUE;
ELSIF NOT FB_waste_pump.PumpWorkingB AND NOT  FB_waste_pump.PumpWorkingF THEN 
	stOutput.bqWastePump:=FALSE;
END_IF

END_PROGRAM

// ---- POUs/050_InkSystem/搅拌_吸废墨/FB/FB_Stirrer.TcPOU
FUNCTION_BLOCK FB_Stirrer
VAR_INPUT
	enable					:BOOL;
	continueTime			:LREAL;//Min   持续时间
	intervalTime			:LREAL;//Min  间隔时间
END_VAR
VAR_OUTPUT
	PumpWorkingF			:BOOL;//正转
	PumpWorkingB			:BOOL;//反转

END_VAR
VAR 
	ton_C:TON;	//   持续时间
	ton_I:TON;	//   持续时间
	step:INT;
	R_trig:R_TRIG;
	F_trig:F_TRIG;
	
END_VAR

R_trig(CLK:=enable , Q=> );
F_trig(CLK:=enable , Q=> );


IF F_trig.Q THEN 
	step:=0;
END_IF

CASE step OF
0://启动
	PumpWorkingF:=FALSE;
	PumpWorkingB:=FALSE;
	ton_C(IN:=FALSE);
	ton_I(IN:=FALSE);
	IF R_trig.Q THEN
	 	step:=10;		
	END_IF	
10://正转
	PumpWorkingF:=TRUE;
	PumpWorkingB:=FALSE;
	ton_I(IN:=FALSE);
	ton_C(IN:=TRUE  , PT:=LREAL_TO_TIME(continueTime*1000*60) , Q=> , ET=> );
	IF ton_C.Q THEN 		
		step:=20;
	END_IF	
20://间隔
	PumpWorkingF:=FALSE;
	PumpWorkingB:=FALSE;
	ton_C(IN:=FALSE);
	ton_I(IN:=TRUE , PT:=LREAL_TO_TIME(intervalTime*1000*60) , Q=> , ET=> );
	IF ton_I.Q THEN 
		step:=30;
	END_IF
30://反转
	PumpWorkingF:=FALSE;
	PumpWorkingB:=TRUE;
	ton_I(IN:=FALSE);
	ton_C(IN:=TRUE  , PT:=LREAL_TO_TIME(continueTime*1000*60) , Q=> , ET=> );
	IF ton_C.Q THEN 		
		step:=40;
	END_IF	
40://间隔
	PumpWorkingF:=FALSE;
	PumpWorkingB:=FALSE;
	ton_C(IN:=FALSE);
	ton_I(IN:=TRUE , PT:=LREAL_TO_TIME(intervalTime*1000*60) , Q=> , ET=> );
	IF ton_I.Q THEN 
		step:=10;
	END_IF

END_CASE

END_FUNCTION_BLOCK

// ---- POUs/030_MediaTransport/TableVacuum/P_TableVacuum.TcPOU
PROGRAM P_TableVacuum
VAR
	FB_TableVacuum:ARRAY[1..number_TableVacuum] OF FB_TableVacuum;
	i:INT;	
	log_ErrorEnum:TabVacErrorEnum;
	log_ID:INT;
END_VAR

ACT_LOG();

FOR i:=1 TO number_TableVacuum DO
	FB_TableVacuum[i](
		vacuum_measured:= GVL_API.stTableVacuum[i].vacuum_measured, 
		vacuum_min:= GVL_API.stTableVacuum[i].vacuum_min, 
		vacuum_max:= GVL_API.stTableVacuum[i].vacuum_max, 
		setpoint:= GVL_API.stTableVacuum[i].setpoint, 
		vacuum_offset_collector:= GVL_API.stTableVacuum[i].vacuum_offset_collector, 
		setpoint_range_pct:= GVL_API.stTableVacuum[i].setpoint_range_pct, 
		vacuum_timeout:= GVL_API.stTableVacuum[i].vacuum_timeout, 
		vacuum_off_timeout:= GVL_API.stTableVacuum[i].vacuum_off_timeout, 
		IO_Error:=P_Modbus_RTU.station_error[1] OR P_Modbus_RTU.station_error[2],
		state=> GVL_API.stTableVacuum[i].state, 
		error_code=> GVL_API.stTableVacuum[i].error_code, 
		Run=> stOutput.bqVacRun[i], 
		error=> GVL_API.stTableVacuum[1].Error, 
		Initialize:= GVL_API.stTableVacuum[i].Initialize, 
		SetVacuumOn:= GVL_API.stTableVacuum[i].SetVacuumOn, 
		SetVacuumOff:= GVL_API.stTableVacuum[i].SetVacuumOff, 
		Setoff:=GVL_API.stTableVacuum[i].Setoff  );
		
END_FOR

ACTION ACT_LOG:
(*************************LOG*******************************************)
log_ID:=300;
//initialize
AlarmActionArray[log_ID+1].AlarmMsg.EN	:=CONCAT('TableVacuum initialize, ',LREAL_TO_STRING(GVL_API.stTableVacuum[1].vacuum_min));
AlarmActionArray[log_ID+1].AlarmMsg.EN	:=CONCAT(AlarmActionArray[log_ID+1].AlarmMsg.EN,', ');
AlarmActionArray[log_ID+1].AlarmMsg.EN	:=CONCAT(AlarmActionArray[log_ID+1].AlarmMsg.EN,
																	LREAL_TO_STRING(GVL_API.stTableVacuum[1].vacuum_max));
AlarmActionArray[log_ID+1].AlarmMsg.EN	:=CONCAT(AlarmActionArray[log_ID+1].AlarmMsg.EN,', ');
AlarmActionArray[log_ID+1].AlarmMsg.EN	:=CONCAT(AlarmActionArray[log_ID+1].AlarmMsg.EN,
																	LREAL_TO_STRING(GVL_API.stTableVacuum[1].setpoint_range_pct));														
fbSetAlarm[log_ID+1](
	InUse:=TRUE , 
	EventId:=log_ID+1 , 
	EventActive:=GVL_API.stTableVacuum[1].Initialize , 
	EventClass:=Alm_EventClass.Event , 
	ToTheLogFile:=TRUE, 
	ToTheHistory:=TRUE , 
 );
 //SetVacuumOn
AlarmActionArray[log_ID+2].AlarmMsg.EN	:=CONCAT('TableVacuum SetVacuumOn, ',LREAL_TO_STRING(GVL_API.stTableVacuum[1].setpoint));
AlarmActionArray[log_ID+2].AlarmMsg.EN	:=CONCAT(AlarmActionArray[log_ID+2].AlarmMsg.EN,', ');
AlarmActionArray[log_ID+2].AlarmMsg.EN	:=CONCAT(AlarmActionArray[log_ID+2].AlarmMsg.EN,
																	LREAL_TO_STRING(GVL_API.stTableVacuum[1].vacuum_timeout));

fbSetAlarm[log_ID+2](
	InUse:=TRUE , 
	EventId:=log_ID+2 , 
	EventActive:=GVL_API.stTableVacuum[1].SetVacuumOn , 
	EventClass:=Alm_EventClass.Event , 
	ToTheLogFile:=TRUE, 
	ToTheHistory:=TRUE , 
 );
 //SetVacuumOff
AlarmActionArray[log_ID+3].AlarmMsg.EN	:=CONCAT('TableVacuum SetVacuumOff, ',LREAL_TO_STRING(GVL_API.stTableVacuum[1].vacuum_off_timeout));

fbSetAlarm[log_ID+3](
	InUse:=TRUE , 
	EventId:=log_ID+3 , 
	EventActive:=GVL_API.stTableVacuum[1].SetVacuumOff , 
	EventClass:=Alm_EventClass.Event , 
	ToTheLogFile:=TRUE, 
	ToTheHistory:=TRUE , 
 );

//ERROR,log_ErrorEnum只能等于一个常数
CASE GVL_API.stTableVacuum[1].error_code  OF
0	:	log_ErrorEnum	:=	0	;
1	:	log_ErrorEnum	:=	1	;
2	:	log_ErrorEnum	:=	2	;
3	:	log_ErrorEnum	:=	3	;
4	:	log_ErrorEnum	:=	4	;
5	:	log_ErrorEnum	:=	5	;
6	:	log_ErrorEnum	:=	6	;
7	:	log_ErrorEnum	:=	7	;
8	:	log_ErrorEnum	:=	8	;
666	:	log_ErrorEnum	:=	666	;


END_CASE

AlarmActionArray[log_ID+9].AlarmMsg.EN	:=CONCAT('TableVacuum Error: ',TO_STRING(log_ErrorEnum));
fbSetAlarm[log_ID+9](
	InUse:=TRUE , 
	EventId:=log_ID+9 , 
	EventActive:=GVL_API.stTableVacuum[1].error_code<>0 AND GVL_API.stTableVacuum[1].error_code<>666   , 
	EventClass:=Alm_EventClass.Alarm , 
	ToTheLogFile:=TRUE, 
	ToTheHistory:=TRUE , 
 );
 
//reset
AlarmActionArray[log_ID+10].AlarmMsg.EN	:=	'TableVacuum Reset ';
fbSetAlarm[log_ID+10](
	InUse:=TRUE , 
	EventId:=log_ID+10 , 
	EventActive:=GVL_API.stTableVacuum[1].Setoff  , 
	EventClass:=Alm_EventClass.Event , 
	ToTheLogFile:=TRUE, 
	ToTheHistory:=TRUE , 
 );
END_ACTION

END_PROGRAM

// ---- POUs/030_MediaTransport/UpDownSlot/P_UpDownSlot.TcPOU
PROGRAM P_UpDownSlot
VAR
	UpDownSlot_S1: FB_UpDownSlotS1;
	UpDownSlot_S2_S6: ARRAY[2..6] OF FB_UpDownSlotS2_S6;
	i:INT;
	log_ErrorEnum:UpDownSlotErrorEnum;
	log_ID:INT;


END_VAR

ACT_LOG();

//S1 急停用2904，S1-S6 只用急停按钮
(***************S1************************************************)
UpDownSlot_S1(
	timeout_up:= GVL_API.stUpDownSlot[1].timeout_up*1000, 
	timeout_down:= GVL_API.stUpDownSlot[1].timeout_down*1000, 
	extra_down_time:= GVL_API.stUpDownSlot[1].extra_down_time*1000, 
	sensor_up:= stInput.biUDS_sensor_up_S[1], 
	sensor_down:= stInput.biUDS_sensor_down_S1, 
	MoveDown_do=> , 
	MoveUp_do=>  , 
	Break=> stOutput.bqS1_Break, 
	anysensor_down=> ,
	state=> GVL_API.stUpDownSlot[1].state, 
	error_code=> GVL_API.stUpDownSlot[1].error_code, 
	error=>GVL_API.stUpDownSlot[1].Error , 
	Initialize:= GVL_API.stUpDownSlot[1].Initialize, 
	MoveDown:= GVL_API.stUpDownSlot[1].MoveDown, 
	MoveUp:= GVL_API.stUpDownSlot[1].MoveUp, 
	SetOff:= GVL_API.stUpDownSlot[1].SetOff );
	
	IF UpDownSlot_S1.MoveDown_do OR  UpDownSlot_S1.MoveUp_do THEN
		stOutput.bqS1_Drive_enabled:=TRUE;
	ELSIF NOT UpDownSlot_S1.MoveDown_do AND NOT   UpDownSlot_S1.MoveUp_do THEN 
		stOutput.bqS1_Drive_enabled:=FALSE;
	END_IF
	
	IF UpDownSlot_S1.MoveDown_do AND NOT  UpDownSlot_S1.MoveUp_do THEN 
		stOutput.bqS1_Forward_Reverse:=FALSE;
	ELSIF NOT UpDownSlot_S1.MoveDown_do AND   UpDownSlot_S1.MoveUp_do THEN 
		stOutput.bqS1_Forward_Reverse:=TRUE;
	END_IF

	GVL_API.stUpDownSlot[1].sensor_up:=stInput.biUDS_sensor_up_S[1];
	GVL_API.stUpDownSlot[1].sensor_down:=UpDownSlot_S1.anysensor_down;
	
(***************S2-S6:************************************************)
FOR i:=2 TO number_UpDownSlot DO
	UpDownSlot_S2_S6[i](
		timeout_up:=GVL_API.stUpDownSlot[i].timeout_up*1000 , 
		timeout_down:= GVL_API.stUpDownSlot[i].timeout_down*1000, 
		sensor_up:= stInput.biUDS_sensor_up_S[i], 
		MoveDown_do=> stOutput.bqUDS_MoveDown_do[i], 
		MoveUp_do=> stOutput.bqUDS_MoveUp_do[i], 
		state=> GVL_API.stUpDownSlot[i].state, 
		error_code=> GVL_API.stUpDownSlot[i].error_code, 
		error=> GVL_API.stUpDownSlot[i].Error, 
		Initialize:= GVL_API.stUpDownSlot[i].Initialize, 
		MoveDown:= GVL_API.stUpDownSlot[i].MoveDown, 
		MoveUp:= GVL_API.stUpDownSlot[i].MoveUp, 
		SetOff:=GVL_API.stUpDownSlot[i].SetOff );
		
		GVL_API.stUpDownSlot[i].sensor_up:=stInput.biUDS_sensor_up_S[i];
END_FOR

ACTION ACT_LOG:
(*************************LOG*******************************************)
log_ID:=320;
(******************s1******************************)
//initialize
AlarmActionArray[log_ID+1].AlarmMsg.EN	:='UpDownSlot1 initialize ';												
fbSetAlarm[log_ID+1](
	InUse:=TRUE , 
	EventId:=log_ID+1 , 
	EventActive:=GVL_API.stUpDownSlot[1].Initialize , 
	EventClass:=Alm_EventClass.Event , 
	ToTheLogFile:=TRUE, 
	ToTheHistory:=TRUE , 
 );
 //MoveDown
AlarmActionArray[log_ID+2].AlarmMsg.EN	:=CONCAT('UpDownSlot1 MoveDown, ',
																	LREAL_TO_STRING(GVL_API.stUpDownSlot[1].timeout_down));
AlarmActionArray[log_ID+2].AlarmMsg.EN	:=CONCAT(AlarmActionArray[log_ID+2].AlarmMsg.EN,', ');
AlarmActionArray[log_ID+2].AlarmMsg.EN	:=CONCAT(AlarmActionArray[log_ID+2].AlarmMsg.EN,
																	LREAL_TO_STRING(GVL_API.stUpDownSlot[1].extra_down_time));

fbSetAlarm[log_ID+2](
	InUse:=TRUE , 
	EventId:=log_ID+2 , 
	EventActive:=GVL_API.stUpDownSlot[1].MoveDown , 
	EventClass:=Alm_EventClass.Event , 
	ToTheLogFile:=TRUE, 
	ToTheHistory:=TRUE , 
 );
 //MoveUp
AlarmActionArray[log_ID+3].AlarmMsg.EN	:=CONCAT('UpDownSlot1 MoveUp, ',
																	LREAL_TO_STRING(GVL_API.stUpDownSlot[1].timeout_up));

fbSetAlarm[log_ID+3](
	InUse:=TRUE , 
	EventId:=log_ID+3 , 
	EventActive:=GVL_API.stUpDownSlot[1].MoveUp , 
	EventClass:=Alm_EventClass.Event , 
	ToTheLogFile:=TRUE, 
	ToTheHistory:=TRUE , 
 );

//ERROR,log_ErrorEnum只能等于一个常数
CASE GVL_API.stUpDownSlot[1].error_code  OF
0	:	log_ErrorEnum	:=	0	;
1	:	log_ErrorEnum	:=	1	;
2	:	log_ErrorEnum	:=	2	;
3	:	log_ErrorEnum	:=	3	;
4	:	log_ErrorEnum	:=	4	;
5	:	log_ErrorEnum	:=	5	;
6	:	log_ErrorEnum	:=	6	;
7	:	log_ErrorEnum	:=	7	;
666	:	log_ErrorEnum	:=	666	;

END_CASE

AlarmActionArray[log_ID+9].AlarmMsg.EN	:=CONCAT('UpDownSlot1 Error: ',TO_STRING(log_ErrorEnum));
fbSetAlarm[log_ID+9](
	InUse:=TRUE , 
	EventId:=log_ID+9 , 
	EventActive:=GVL_API.stUpDownSlot[1].error_code<>0  AND GVL_API.stUpDownSlot[1].error_code<>666, 
	EventClass:=Alm_EventClass.Alarm , 
	ToTheLogFile:=TRUE, 
	ToTheHistory:=TRUE , 
 );
 
//reset
AlarmActionArray[log_ID+10].AlarmMsg.EN	:=	'UpDownSlot1 Reset ';
fbSetAlarm[log_ID+10](
	InUse:=TRUE , 
	EventId:=log_ID+10 , 
	EventActive:=GVL_API.stUpDownSlot[1].SetOff  , 
	EventClass:=Alm_EventClass.Event , 
	ToTheLogFile:=TRUE, 
	ToTheHistory:=TRUE , 
 );
 
 
(******************s2-s6******************************)
FOR i:=2 TO number_UpDownSlot DO
//initialize
AlarmActionArray[log_ID+10*i+1].AlarmMsg.EN	:=CONCAT('UpDownSlot',
																			INT_TO_STRING(i));
AlarmActionArray[log_ID+10*i+1].AlarmMsg.EN	:=CONCAT(AlarmActionArray[log_ID+10*i+1].AlarmMsg.EN,
																			' initialize');												
fbSetAlarm[log_ID+10*i+1](
	InUse:=TRUE , 
	EventId:=log_ID+10*i+1 , 
	EventActive:=GVL_API.stUpDownSlot[i].Initialize , 
	EventClass:=Alm_EventClass.Event , 
	ToTheLogFile:=TRUE, 
	ToTheHistory:=TRUE , 
 );
 //MoveDown
 AlarmActionArray[log_ID+10*i+2].AlarmMsg.EN	:=CONCAT('UpDownSlot',
																			INT_TO_STRING(i));
AlarmActionArray[log_ID+10*i+2].AlarmMsg.EN	:=CONCAT(AlarmActionArray[log_ID+10*i+2].AlarmMsg.EN,
																			' MoveDown');
AlarmActionArray[log_ID+10*i+2].AlarmMsg.EN	:=CONCAT(AlarmActionArray[log_ID+10*i+2].AlarmMsg.EN,', ');	
AlarmActionArray[log_ID+10*i+2].AlarmMsg.EN	:=CONCAT(AlarmActionArray[log_ID+10*i+2].AlarmMsg.EN,
																	LREAL_TO_STRING(GVL_API.stUpDownSlot[i].timeout_down));

fbSetAlarm[log_ID+10*i+2](
	InUse:=TRUE , 
	EventId:=log_ID+10*i+2 , 
	EventActive:=GVL_API.stUpDownSlot[i].MoveDown , 
	EventClass:=Alm_EventClass.Event , 
	ToTheLogFile:=TRUE, 
	ToTheHistory:=TRUE , 
 );
 //MoveUp
AlarmActionArray[log_ID+10*i+3].AlarmMsg.EN	:=CONCAT('UpDownSlot',
																			INT_TO_STRING(i));
AlarmActionArray[log_ID+10*i+3].AlarmMsg.EN	:=CONCAT(AlarmActionArray[log_ID+10*i+3].AlarmMsg.EN,
																			' MoveUp');
AlarmActionArray[log_ID+10*i+3].AlarmMsg.EN	:=CONCAT(AlarmActionArray[log_ID+10*i+3].AlarmMsg.EN,', ');	
AlarmActionArray[log_ID+10*i+3].AlarmMsg.EN	:=CONCAT(AlarmActionArray[log_ID+10*i+3].AlarmMsg.EN,
																	LREAL_TO_STRING(GVL_API.stUpDownSlot[i].timeout_up));

fbSetAlarm[log_ID+10*i+3](
	InUse:=TRUE , 
	EventId:=log_ID+10*i+3 , 
	EventActive:=GVL_API.stUpDownSlot[i].MoveUp , 
	EventClass:=Alm_EventClass.Event , 
	ToTheLogFile:=TRUE, 
	ToTheHistory:=TRUE , 
 );

//ERROR,log_ErrorEnum只能等于一个常数
CASE GVL_API.stUpDownSlot[i].error_code  OF
0	:	log_ErrorEnum	:=	0	;
1	:	log_ErrorEnum	:=	1	;
2	:	log_ErrorEnum	:=	2	;
3	:	log_ErrorEnum	:=	3	;
4	:	log_ErrorEnum	:=	4	;
5	:	log_ErrorEnum	:=	5	;
6	:	log_ErrorEnum	:=	6	;
7	:	log_ErrorEnum	:=	7	;
666	:	log_ErrorEnum	:=	666	;


END_CASE
AlarmActionArray[log_ID+10*i+9].AlarmMsg.EN	:=CONCAT('UpDownSlot',INT_TO_STRING(i));
AlarmActionArray[log_ID+10*i+9].AlarmMsg.EN	:=CONCAT(AlarmActionArray[log_ID+10*i+9].AlarmMsg.EN,
																			' Error: ');
AlarmActionArray[log_ID+10*i+9].AlarmMsg.EN	:=CONCAT(AlarmActionArray[log_ID+10*i+9].AlarmMsg.EN,
																			TO_STRING(log_ErrorEnum));																			

fbSetAlarm[log_ID+10*i+9](
	InUse:=TRUE , 
	EventId:=log_ID+10*i+9 , 
	EventActive:=GVL_API.stUpDownSlot[i].error_code<>0 AND GVL_API.stUpDownSlot[i].error_code<>666 , 
	EventClass:=Alm_EventClass.Alarm , 
	ToTheLogFile:=TRUE, 
	ToTheHistory:=TRUE , 
 );
 
//reset
AlarmActionArray[log_ID+10*i+10].AlarmMsg.EN	:=CONCAT('UpDownSlot',
																			INT_TO_STRING(i));
AlarmActionArray[log_ID+10*i+10].AlarmMsg.EN	:=CONCAT(AlarmActionArray[log_ID+10*i+10].AlarmMsg.EN,
																			' Reset');		

fbSetAlarm[log_ID+10*i+10](
	InUse:=TRUE , 
	EventId:=log_ID+10*i+10 , 
	EventActive:=GVL_API.stUpDownSlot[i].SetOff  , 
	EventClass:=Alm_EventClass.Event , 
	ToTheLogFile:=TRUE, 
	ToTheHistory:=TRUE , 
 );
END_FOR
 (*************em-stop*     *************
 AlarmActionArray[399].AlarmMsg.EN	:='UpDownSlot Error: emergency_error';																		

fbSetAlarm[399](
	InUse:=TRUE , 
	EventId:=399 , 
	EventActive:=GVL_API.stUpDownSlot[i].error_code=666 , 
	EventClass:=Alm_EventClass.Alarm , 
	ToTheLogFile:=TRUE, 
	ToTheHistory:=TRUE , 
 );
*)
END_ACTION

END_PROGRAM

// ---- POUs/010_Motion/MotionBase/PTP/Axis_PTP_CoE.TcPOU
FUNCTION_BLOCK Axis_PTP_CoE
VAR_INPUT	
	Ref:					AXIS_REF;
	IO:						Axis_IO;
	mcJog:					MC_Jog;
	mcHome:					MC_Home;
	mcMoveAbsolute:			MC_MoveAbsolute;
	mcMoveRelative:			MC_MoveRelative;
	mcMoveVelocity:			MC_MoveVelocity;	
	mcPower:				MC_Power;
	mcReset:				MC_Reset;
	mcStop:					MC_Stop;
	mcReadStatus			:MC_ReadStatus;
	mcSetPostion			:MC_SetPosition;

	Target					:LREAL;
	Velo					:LREAL;
	Jerk					:LREAL ;
	Acc						:LREAL ;
	Dec						:LREAL ;
	
	Execute					:BOOL;
	power_do				:BOOL;
	stop_do					:BOOL;
	Reset_do				:BOOL;
	JogF,JogB				:BOOL;
	MoveRel_do				:BOOL;
	MoveAbs_do				:BOOL;

END_VAR
VAR_OUTPUT
	Done:					BOOL;(*功能块执行完成状态*)
	Busy: 					BOOL;(*功能块正在执行状态*)
	Active:					BOOL;
	CommandAborted:			BOOL;
	Error:					BOOL;
	ErrorID:				UDINT;
END_VAR

ACTION aHome:
(*
TYPE MC_HomingMode :
(
	MC_DefaultHoming,		(* default homing as defined in the SystemManager encoder parameters *)
	MC_AbsSwitch, 		(* not implemented - Absolute Switch homing plus Limit switches *)
	MC_LimitSwitch, 		(* not implemented - Homing against Limit switches *)
	MC_RefPulse, 		(* not implemented - Homing using encoder Reference Pulse "Zero Mark" *)
	MC_Direct, 		(* Static Homing forcing position from user reference *)
	MC_Absolute, 		(* not implemented - Static Homing forcing position from absolute encoder *)
	MC_Block, 		(* not implemented - Homing against hardware parts blocking movement *)
	MC_ForceCalibration, 	(* set the calibration flag without performing any motion or changing the position *)
	MC_ResetCalibration  	(* resets the calibration flag without performing any motion or changing the position *)
);
END_TYPE

*)


mcHome(
	Axis:=Ref , 
	Execute:=Execute , 
	Position:= , 
	HomingMode:= , 
	BufferMode:= , 
	Options:= , 
	bCalibrationCam:= , 
	Done=> , 
	Busy=> , 
	Active=> , 
	CommandAborted=> , 
	Error=> , 
	ErrorID=> );
END_ACTION

ACTION aJogB:
mcJog(
	JogForward:= 	FALSE,
	JogBackwards:= 	Execute,
	Mode:= 			MC_JOGMODE_CONTINOUS,
	Position:= 		,
	Velocity:= 		Velo,
	Acceleration:= 	Acc,
	Deceleration:= 	Dec,
	Jerk:= 			Jerk,
	Axis:= 			Ref,
	Busy=> 			Busy,
	Active=> 		Active,
	CommandAborted=> CommandAborted,
	Error=> 		Error,
	ErrorID=> 		ErrorID
	);
END_ACTION

ACTION aJogF:
mcJog(
	JogForward:= 	Execute,
	JogBackwards:= 	FALSE,
	Mode:= 			MC_JOGMODE_CONTINOUS,
	Position:= 		,
	Velocity:= 		Velo,
	Acceleration:= 	Acc,
	Deceleration:= 	Dec,
	Jerk:= 			Jerk,
	Axis:= 			Ref,
	Busy=> 			Busy,
	Active=> 		Active,
	CommandAborted=> CommandAborted,
	Error=> 		Error,
	ErrorID=> 		ErrorID
	);
END_ACTION

ACTION aManualJOG:
(*
TYPE E_JogMode :
(
	MC_JOGMODE_STANDARD_SLOW, (* motion with standard jog parameters for slow motion *)
	MC_JOGMODE_STANDARD_FAST, (* motion with standard jog parameters for fast motion *)
	MC_JOGMODE_CONTINOUS,     (* axis moves as long as the jog button is pressed using parameterized dynamics *)
	MC_JOGMODE_INCHING,       (* axis moves for a certain relative distance *)
	MC_JOGMODE_INCHING_MODULO (* axis moves for a certain relative distance - stop position is rounded to the distance value *)
);
END_TYPE

*)

mcJog(
	JogForward:= 	JogF,
	JogBackwards:= 	JogB,
	Mode:= 			MC_JOGMODE_CONTINOUS,
	Position:= 		,
	Velocity:= 		Velo,
	Acceleration:= 	Acc,
	Deceleration:= 	Dec,
	Jerk:= 			Jerk,
	Axis:= 			Ref,
	Busy=> 			,
	Active=> 		,
	CommandAborted=> ,
	Error=> 		,
	ErrorID=> 		
	);
END_ACTION

ACTION aManualMoveAbs:
mcMoveAbsolute(
	Execute:= 		IO.btManualABS,
	Position:= 		Target,
	Velocity:= 		Velo,
	Acceleration:= 	Acc,
	Deceleration:= 	Dec,
	Jerk:= 			Jerk,
	Axis:= 			Ref,
	Done=> 			,
	Busy=> 			,
	Active=> 		,
	CommandAborted=> ,
	Error=> 		Error,
	ErrorID=> 		ErrorID
	);
END_ACTION

ACTION aMoveAbs:
mcMoveAbsolute(
	Execute:= 		MoveAbs_do,
	Position:= 		Target,
	Velocity:= 		Velo,
	Acceleration:= 	Acc,
	Deceleration:= 	Dec,
	Jerk:= 			Jerk,
	Axis:= 			Ref,
	Done=> 			,
	Busy=> 			,
	Active=> 		Active,
	CommandAborted=> CommandAborted,
	Error=> 		Error,
	ErrorID=> 		ErrorID
	);
END_ACTION

ACTION aMoveOff:
(*关轴*)
mcHome(
	Execute:= 		FALSE,
	Axis:= 			Ref,
	);

mcJog(
	JogForward:= 	FALSE,
	JogBackwards:= 	FALSE,
	Axis:= 			Ref,
	);

mcMoveAbsolute(
	Execute:= 		FALSE,
	Axis:= 			Ref,
	);

mcMoveRelative(
	Execute:= 		FALSE,
	Axis:= 			Ref,
	);

mcMoveVelocity(
	Execute:= 		FALSE,
	Axis:= 			Ref,
	);

Done:=FALSE;
Busy:=FALSE;
Active:=FALSE;
CommandAborted:=FALSE;
Error:=FALSE;
END_ACTION

ACTION aMoveRel:
mcMoveRelative(
	Execute:= 		MoveRel_do,
	Distance:= 		Target,
	Velocity:= 		Velo,
	Acceleration:= 	Acc,
	Deceleration:= 	Dec,
	Jerk:= 			Jerk,
	Axis:= 			Ref,
	Done=> 			Done,
	Busy=> 			Busy,
	Active=> 		Active,
	CommandAborted=> CommandAborted,
	Error=> 		Error,
	ErrorID=> 		ErrorID
	);
END_ACTION

ACTION aMoveVel:
mcMoveVelocity(
	Execute:= 		Execute,
	Direction:= 	,
	Velocity:= 		Velo,
	Acceleration:= 	Acc,
	Deceleration:= 	Dec,
	Jerk:= 			Jerk,
	Axis:= 			Ref,
	InVelocity=> 	Done,
	Busy=> 			Busy,
	Active=> 		Active,
	CommandAborted=> CommandAborted,
	Error=> 		Error,
	ErrorID=> 		ErrorID );
END_ACTION

ACTION aPower:
mcPower(
	Enable:= power_do		,
	Enable_Positive:=TRUE 	,
	Enable_Negative:=TRUE	,
	Override:= 		,
	BufferMode:= 	,
	Axis:= 			Ref,
	Status=> 		,
	Busy=> 			,
	Active=> 		,
	Error=> 		Error,
	ErrorID=> 		ErrorID
	);
END_ACTION

ACTION aReadStatus:
mcReadStatus(
	Axis:=Ref , 
	Enable:=TRUE , 
	Valid=> , 
	Busy=> , 
	Error=> , 
	ErrorID=> , 
	ErrorStop=> , 
	Disabled=> , 
	Stopping=> , 
	StandStill=> , 
	DiscreteMotion=> , 
	ContinuousMotion=> , 
	SynchronizedMotion=> , 
	Homing=> , 
	ConstantVelocity=> , 
	Accelerating=> , 
	Decelerating=> , 
	Status=> );
END_ACTION

ACTION aReset:
Ref.ReadStatus();(*读取轴状态*);

(*复位*)
mcReset(
	Execute:= 	Reset_do
				(*AND Ref.Status.Error*),
	Axis:= 		Ref,
	);
mcSetPostion(
	Axis:=Ref , 
	Execute:=Reset_do , 
	Position:= , 
	Mode:= , 
	Options:= , 
	Done=> , 
	Busy=> , 
	Error=> , 
	ErrorID=> );
IF (mcReset.Busy OR mcReset.Done) AND mcSetPostion.Done THEN 
	Reset_do:=FALSE;
END_IF

(**)
END_ACTION

ACTION aSetPostion:
mcSetPostion(
	Axis:=Ref , 
	Execute:=Reset_do , 
	Position:=0 , 
	Mode:= , 
	Options:= , 
	Done=> , 
	Busy=> , 
	Error=> , 
	ErrorID=> );
END_ACTION

ACTION aStop:
IF Execute THEN 
	aMoveOff();
END_IF


mcStop(
	Execute:= 		stop_do,
	Deceleration:= 	Dec,
	Jerk:= 			Jerk,
	Options:= 		,
	Axis:= 			Ref,
	Done=> 			Done,
	Busy=> 			Busy,
	Active=> 		Active,
	CommandAborted=> CommandAborted,
	Error=> 		Error,
	ErrorID=> 		ErrorID
	);
IF mcStop.Done OR mcStop.Busy  THEN 
	stop_do:=FALSE;
END_IF
END_ACTION

END_FUNCTION_BLOCK

// ---- POUs/010_Motion/P_Motion.TcPOU
PROGRAM P_Motion
VAR

END_VAR

P_FastScan();
P_Z_Axis();
P_SlowScan();

END_PROGRAM

// ---- POUs/060_UVLed/FB/FB_UVLed_L.TcPOU
(**************1个LED灯*************************)
FUNCTION_BLOCK FB_UVLed_L
VAR_INPUT
	single_double			:BOOL;//"Indicates unidirectional printing.TRUE IF the print is unidirectional, otherwise FALSE FOR bi-directional printing.
	initial_print_position	:INT;//"Indicates the initial print position: 0:from_home, 1:to_home."
	uv_power_leading		:DINT;//% "(leadingPower ConfigurePower-Settings method)Power to apply to leading LEDs of the UVUnit"
	uv_power_trailing		:DINT;//% "(trailingPower ConfigurePower-Settings method)Power to apply to trailing LEDs of the UVUnit"
	uvStart					:LREAL;//mm "Position in micron where to start/stop curing depending on the direction (left/right)."
	uvEnd					:LREAL;//mm "Position in micron where to start/stop curing depending on the direction (left/right)"
	ahead_pos				:LREAL:=100;//UV开灯提前
	delay_pos				:LREAL:=100;//UV关闭延迟
	parts					:BYTE;
	
	Encoder					:LREAL;
	Moving					:BOOL;//fs MOVING
	FS_Direction_N			:BOOL;//反向
	FS_Direction_P			:BOOL;//正向
	UVError					:BOOL;
	IO_Error				:BOOL;
	UVisRemote				:BOOL;
END_VAR
VAR_OUTPUT
	state				:INT;
	error_code			:INT;
	uv_power			:DINT;//一个UV灯内 分段功率
	set_prats			:BYTE;//
	initialized			:BOOL;
	settings_applide		:BOOL;
	curing_started	:BOOL;
	curing_stopped	:BOOL;
	error					:BOOL;
	off					:BOOL;
END_VAR
VAR
	step				:INT;
	unidirection		:BOOL;//单向
	bidirectiona		:BOOL;//双向
	from_home			:BOOL;//Printing starts from the home position
	to_home				:BOOL;//Printing starts towards the home position
	error_trig1,error_trig2:Tc2_Standard.R_TRIG;
	uvStart_temp		:LREAL;//因UV灯有延迟，提前量
	uvEnd_temp			:LREAL;//因UV灯有延迟，提前量
	ton1:Tc2_Standard.TON;
END_VAR
VAR_IN_OUT
	Initialize				:BOOL;
	ConfigurePowerSettings	:BOOL;
	ConfigurePositions		:BOOL;
	StopCuring				:BOOL;
	SetOff					:BOOL;
END_VAR

set_prats:=parts;

(***************因UV灯有延迟，提前量****************************)
	uvStart_temp:=uvStart-ahead_pos;
	uvEnd_temp:=uvEnd+delay_pos;

CASE step OF
0://waiting
	IF Initialize THEN 
		step:=5;	
	ELSIF ConfigurePowerSettings THEN 
		step:=20;	
	ELSIF ConfigurePositions THEN 
		step:=40;
	ELSIF ConfigurePowerSettings THEN 
		step:=10;
	ELSIF StopCuring THEN 
		step:=40;
	ELSIF SetOff OR GVL.Reset THEN 
		step:=200;
	ELSIF state=UVLedStateEnum.ready_for_curing AND Moving THEN 
		step:=50;
	END_IF
	(******************状态自复位***************************)
	ton1(IN:=initialized OR  settings_applide OR  curing_started OR  curing_stopped 
				OR error OR  off , PT:=State_reset_time , Q=> , ET=> );
	IF ton1.Q THEN 
		initialized:=FALSE;
		settings_applide:=FALSE;
		curing_started:=FALSE;
		curing_stopped:=FALSE;
		error:=FALSE;
		off:=FALSE;
	END_IF
	
5://off
	state:=UVLedStateEnum.off;
	error_code:=UVLedErrorEnum.no_error;	
	uv_power:=0;
	
	ConfigurePowerSettings	:=FALSE;
	ConfigurePositions		:=FALSE;
	StopCuring				:=FALSE;
	SetOff					:=FALSE;
	bidirectiona			:=FALSE;
	from_home				:=FALSE;
	
	IF Initialize  THEN 
		Initialize:=FALSE;	
		state:=UVLedStateEnum.initializing;	
		step:=6;		
	END_IF
6://
	IF UVisRemote THEN 
		step:=10;	
	END_IF
10://initializing	
	initialized:=TRUE;
	state:=UVLedStateEnum.ready;	
	settings_applide:=FALSE;
	curing_started:=FALSE;
	curing_stopped:=FALSE;
	off:=FALSE;
	step:=0;
20://ready	
	IF 	ConfigurePowerSettings THEN
		ConfigurePowerSettings:=FALSE; 
		IF single_double THEN 
			unidirection:=TRUE;
			bidirectiona:=FALSE;
		ELSE
			unidirection:=FALSE;
			bidirectiona:=TRUE;
		END_IF
		IF initial_print_position=1 THEN 
			to_home:=TRUE;
			from_home:=FALSE;
		ELSIF initial_print_position=0 THEN 
			to_home:=FALSE;
			from_home:=TRUE;
		END_IF		
		state:=UVLedStateEnum.applying_settings;
		step:=30;
	END_IF
	IF SetOff THEN	
		step :=200;
	END_IF
30://applying_settings
	ConfigurePowerSettings:=FALSE;	
	uv_power:=0;
	state:=UVLedStateEnum.settings_applied;
	settings_applide:=TRUE;
	step:=0;
40://settings_applied	
	IF 	ConfigurePositions THEN 
		ConfigurePositions:=FALSE;
		IF uvStart>0 AND uvEnd>0   THEN 
			state:=UVLedStateEnum.ready_for_curing;
			step:=0;
		END_IF	
	END_IF
	IF StopCuring THEN 
		StopCuring:=FALSE;
		state:=UVLedStateEnum.ready;
		step:=0;
	END_IF
50://ready_for_curing
	//IF is_printing THEN 
		IF bidirectiona THEN 
			step:=60;
		ELSIF unidirection THEN 
			IF from_home THEN 
				step:=70;
			ELSIF to_home THEN 
				step:=80;
			END_IF
		END_IF
	//END_IF
60://bidirectiona   双向
	IF FS_Direction_P THEN 	//向右
		IF Encoder>=uvStart_temp  AND Encoder<=uvEnd_temp THEN    //左灯
			 uv_power:=uv_power_trailing;	
			curing_started :=TRUE;
		ELSE uv_power:=0;
		END_IF
		IF Encoder>uvEnd_temp  THEN  //结束
			curing_started :=FALSE;
			curing_stopped:=TRUE;
			step:=30;
		END_IF
	ELSIF FS_Direction_N THEN 
		IF Encoder>=uvStart_temp  AND Encoder<=uvEnd_temp THEN    //左灯
			 uv_power:=uv_power_leading;
			 curing_started :=TRUE;
		ELSE uv_power:=0;
		END_IF
		IF Encoder<uvStart_temp  THEN  //结束
			curing_started :=FALSE;
			curing_stopped:=TRUE;
			step:=30;
		END_IF
	END_IF
	
	IF uv_power<>0  THEN 
		state:=UVLedStateEnum.curing;
	END_IF

	(*******范围内小车不运动*******)
	IF (Encoder>=uvStart_temp AND Encoder <=uvEnd_temp) AND NOT Moving (*OR NOT is_printing *) THEN 
		uv_power:=0;
		curing_stopped:=TRUE;
		step:=30; 
	END_IF
70://unidirection/from_home
	IF FS_Direction_P THEN 
		IF Encoder>=uvStart_temp  AND Encoder<=uvEnd_temp THEN    //左灯
			 uv_power:=uv_power_trailing;
			  curing_started :=TRUE;
		ELSE uv_power:=0;
		END_IF
		IF Encoder>uvEnd_temp  THEN  //结束
			curing_started :=FALSE;
			curing_stopped:=TRUE;
			step:=30;
		END_IF				
	END_IF
	
	IF uv_power<>0  THEN 
		state:=UVLedStateEnum.curing;
	END_IF
	IF FS_Direction_N THEN 
		uv_power:=0;
		curing_stopped:=TRUE;
		step:=30; 
	END_IF
	(*******范围内小车不运动******)
	IF (Encoder>=uvStart_temp AND Encoder <=uvEnd_temp) AND NOT Moving (*OR NOT is_printing *) THEN 
		uv_power:=0;
		curing_stopped:=TRUE;
		step:=30; 
	END_IF

80://unidirection/to_home
	IF FS_Direction_N THEN 
		IF Encoder>=uvStart_temp  AND Encoder<=uvEnd_temp THEN    //左灯
			 uv_power:=uv_power_leading;
			 curing_started :=TRUE;
		ELSE uv_power:=0;
		END_IF
		IF Encoder<uvStart_temp  THEN  //结束
			curing_started :=FALSE;
			curing_stopped:=TRUE;
			step:=30;
		END_IF	
	END_IF
	
	IF uv_power<>0  THEN 
		state:=UVLedStateEnum.curing;
	END_IF
	IF FS_Direction_P THEN 
		uv_power:=0;
		curing_stopped:=TRUE;
		step:=30; 
	END_IF
	(*******范围内小车不运动*******)
	IF (Encoder>=uvStart_temp AND Encoder <=uvEnd_temp) AND NOT Moving (*OR NOT is_printing*)  THEN 
		uv_power:=0;
		curing_stopped:=TRUE;
		step:=30; 
	END_IF
100://error
	state:=UVLedStateEnum.error;
	error:=TRUE;
	uv_power:=0;
	step:=0; 
	IF SetOff OR GVL.Reset THEN
		SetOff:=FALSE; 	
		step :=200;
	END_IF
200://seting_off	
	SetOff:=FALSE; 
	state:=UVLedStateEnum.setting_off;
	error_code:=UVLedErrorEnum.no_error;
	uv_power:=0;
	off:=TRUE;
	state:=UVLedStateEnum.off;
	step:=0;
END_CASE
IF SetOff OR GVL.Reset THEN 
	step:=200;
END_IF

(*****************ERROR**************************************)
IF 	state<>UVLedStateEnum.setting_off AND state<>UVLedStateEnum.off AND state<>UVLedStateEnum.error THEN 
	error_trig1(CLK:=UVError AND state<>UVLedStateEnum.off , Q=> );
	error_trig2(CLK:=IO_Error AND state<>UVLedStateEnum.off , Q=> );
	IF GVL.Emstop_SAFE THEN 
		error_code:=UVLedErrorEnum.emergency_error;
		step:=100;
	ELSIF error_trig1.Q THEN 
		error_code:=UVLedErrorEnum.abnormal_temperature;
		step:=100;
	ELSIF error_trig2.Q THEN 
		error_code:=UVLedErrorEnum.unknown_error;
		step:=100;
	END_IF
END_IF

	(*******只要速度低于值，就不开灯*****)
IF ABS( Axis[FastScan].Ref.NcToPlc.ActVelo)<=10 THEN
	uv_power:=0;	
END_IF

END_FUNCTION_BLOCK

// ---- POUs/060_UVLed/FB/FB_UVLed_R.TcPOU
(**************1个LED灯*************************)
FUNCTION_BLOCK FB_UVLed_R
VAR_INPUT
	single_double			:BOOL;//"Indicates unidirectional printing.TRUE IF the print is unidirectional, otherwise FALSE FOR bi-directional printing.
	initial_print_position	:INT;//"Indicates the initial print position: 0:from_home, 1:to_home."
	uv_power_leading		:DINT;//% "(leadingPower ConfigurePower-Settings method)Power to apply to leading LEDs of the UVUnit"
	uv_power_trailing		:DINT;//% "(trailingPower ConfigurePower-Settings method)Power to apply to trailing LEDs of the UVUnit"
	uvStart					:LREAL;//um "Position in micron where to start/stop curing depending on the direction (left/right)."	
	uvEnd					:LREAL;//mm "Position in micron where to start/stop curing depending on the direction (left/right)"
	ahead_pos				:LREAL:=100;//因YV灯有延迟，提前量uvEnd					:LREAL;//um "Position in micron where to start/stop curing depending on the direction (left/right)"	
	delay_pos				:LREAL:=100;//UV关闭延迟
	parts					:BYTE;
	
	Encoder					:LREAL;
	Moving					:BOOL;//fs MOVING
	FS_Direction_N			:BOOL;//反向
	FS_Direction_P			:BOOL;//正向
	//is_printing				:BOOL;
	UVError					:BOOL;
	IO_Error				:BOOL;
	UVisRemote				:BOOL;
END_VAR
VAR_OUTPUT
	state				:INT;
	error_code				:INT;
	uv_power		:DINT;//一个UV灯内 分段功率
	set_prats				:BYTE;//
	initialized			:BOOL;
	settings_applide		:BOOL;
	curing_started	:BOOL;
	curing_stopped	:BOOL;
	error					:BOOL;
	off					:BOOL;
	
END_VAR
VAR
	step				:INT;
	unidirection		:BOOL;//单向
	bidirectiona		:BOOL;//双向
	from_home			:BOOL;//Printing starts from the home position
	to_home				:BOOL;//Printing starts towards the home position
	error_trig1,error_trig2:Tc2_Standard.R_TRIG;
	uvStart_temp		:LREAL;
	uvEnd_temp			:LREAL;
	ton1:Tc2_Standard.TON;
END_VAR
VAR_IN_OUT
	Initialize				:BOOL;
	ConfigurePowerSettings	:BOOL;
	ConfigurePositions		:BOOL;
	StopCuring				:BOOL;
	SetOff					:BOOL;
END_VAR

set_prats:=parts;

(***************因YV灯有延迟，提前量****************************)
	uvStart_temp:=uvStart-ahead_pos;
	uvEnd_temp:=uvEnd+delay_pos;

CASE step OF
0://waiting
	IF Initialize THEN 
		step:=5;	
	ELSIF ConfigurePowerSettings THEN 
		step:=20;	
	ELSIF ConfigurePositions THEN 
		step:=40;
	ELSIF ConfigurePowerSettings THEN 
		step:=10;
	ELSIF StopCuring THEN 
		step:=40;
	ELSIF SetOff OR GVL.Reset THEN 
		step:=200;
	ELSIF state=UVLedStateEnum.ready_for_curing AND Moving THEN 
		step:=50;
	END_IF
	(******************状态自复位***************************)
	ton1(IN:=initialized OR  settings_applide OR  curing_started OR  curing_stopped 
				OR error OR  off , PT:=State_reset_time , Q=> , ET=> );
	IF ton1.Q THEN 
		initialized:=FALSE;
		settings_applide:=FALSE;
		curing_started:=FALSE;
		curing_stopped:=FALSE;
		error:=FALSE;
		off:=FALSE;
	END_IF
	
5://off
	state:=UVLedStateEnum.off;
	error_code:=UVLedErrorEnum.no_error;	
	uv_power:=0;
	
	ConfigurePowerSettings	:=FALSE;
	ConfigurePositions		:=FALSE;
	StopCuring				:=FALSE;
	SetOff					:=FALSE;
	bidirectiona			:=FALSE;
	from_home				:=FALSE;
	
	IF Initialize THEN 
		Initialize:=FALSE;
		state:=UVLedStateEnum.initializing;	
		step:=6;		
	END_IF
6://
	IF UVisRemote THEN 
		step:=10;	
	END_IF	
10://initializing	
	initialized:=TRUE;
	state:=UVLedStateEnum.ready;
	settings_applide:=FALSE;
	curing_started:=FALSE;
	curing_stopped:=FALSE;
	off:=FALSE;
	step:=0;
20://ready
	IF 	ConfigurePowerSettings THEN
		ConfigurePowerSettings:=FALSE; 
		IF single_double THEN 
			unidirection:=TRUE;
			bidirectiona:=FALSE;
		ELSE
			unidirection:=FALSE;
			bidirectiona:=TRUE;
		END_IF
		IF initial_print_position=1 THEN 
			to_home:=TRUE;
			from_home:=FALSE;
		ELSIF initial_print_position=0 THEN 
			to_home:=FALSE;
			from_home:=TRUE;
		END_IF
		state:=UVLedStateEnum.applying_settings;
		step:=30;
	END_IF
	IF SetOff OR GVL.Reset THEN	
		step :=200;
	END_IF
30://applying_settings
	ConfigurePowerSettings:=FALSE;	
	uv_power:=0;
	state:=UVLedStateEnum.settings_applied;
	settings_applide:=TRUE;
	step:=0;
40://settings_applied
	IF 	ConfigurePositions THEN 
		ConfigurePositions:=FALSE;
		IF uvStart>0 AND uvEnd>0   THEN 
			state:=UVLedStateEnum.ready_for_curing;
			step:=0;
		END_IF	
	END_IF
	IF StopCuring THEN 
		StopCuring:=FALSE;
		state:=UVLedStateEnum.ready;
		step:=0;
	END_IF
50://ready_for_curing
	//IF is_printing THEN 
		IF bidirectiona THEN 
			step:=60;
		ELSIF unidirection THEN 
			IF from_home THEN 
				step:=70;
			ELSIF to_home THEN 
				step:=80;
			END_IF
		END_IF
	//END_IF
60://bidirectiona   双向
	IF FS_Direction_P THEN 	//向右
		IF Encoder>=uvStart_temp  AND Encoder<=uvEnd_temp THEN    //右灯
			 uv_power:=uv_power_leading;
			 curing_started :=TRUE;
		ELSE uv_power:=0;
		END_IF	
		IF Encoder>uvEnd_temp  THEN  //结束
			curing_started :=FALSE;
			curing_stopped:=TRUE;
			step:=30;
		END_IF
	ELSIF FS_Direction_N THEN 
		IF Encoder>=uvStart_temp  AND Encoder<=uvEnd_temp THEN    //右灯
			 uv_power:=uv_power_trailing;
			 curing_started :=TRUE;
		ELSE uv_power:=0;
		END_IF
		IF Encoder<uvStart_temp  THEN  //结束
			curing_started :=FALSE;
			curing_stopped:=TRUE;
			step:=30;
		END_IF
	END_IF
	
	IF uv_power<>0 THEN 
		state:=UVLedStateEnum.curing;
	END_IF

	(*******范围内小车不运动*******)
	IF (Encoder>=uvStart_temp AND Encoder <=uvEnd_temp) AND NOT Moving (*OR NOT is_printing*)  THEN 
		uv_power:=0;
		curing_stopped:=TRUE;
		step:=30; 
	END_IF
70://unidirection/from_home
	IF FS_Direction_P THEN 
		IF Encoder>=uvStart_temp  AND Encoder<=uvEnd_temp THEN    //右灯
			 uv_power:=uv_power_leading;
			 curing_started :=TRUE;
		ELSE uv_power:=0;
		END_IF
		IF Encoder>uvEnd_temp  THEN  //结束
			curing_started :=FALSE;
			curing_stopped:=TRUE;
			step:=30;
		END_IF				
	END_IF
	
	IF uv_power<>0  THEN 
		state:=UVLedStateEnum.curing;
	END_IF
	IF FS_Direction_N THEN 
		uv_power:=0;
		curing_stopped:=TRUE;
		step:=30; 
	END_IF
	(*******范围内小车不运动*******)
	IF (Encoder>=uvStart_temp AND Encoder <=uvEnd_temp) AND NOT Moving (* OR NOT is_printing*)  THEN 
		uv_power:=0;
		curing_stopped:=TRUE;
		step:=30; 
	END_IF
	
80://unidirection/to_home
	IF FS_Direction_N THEN 
		IF Encoder>=uvStart_temp  AND Encoder<=uvEnd_temp THEN    //右灯
			 uv_power:=uv_power_trailing;
			 curing_started :=TRUE;
		ELSE uv_power:=0;
		END_IF
		IF Encoder<uvStart_temp  THEN  //结束
			curing_started :=FALSE;
			curing_stopped:=TRUE;
			step:=30;
		END_IF	
	END_IF
	
	IF uv_power<>0 THEN 
		state:=UVLedStateEnum.curing;
	END_IF
	IF FS_Direction_P THEN 
		uv_power:=0;
		curing_stopped:=TRUE;
		step:=30; 
	END_IF
	(*******范围内小车不运动*******)
	IF (Encoder>=uvStart_temp AND Encoder <=uvEnd_temp) AND NOT Moving  (*OR NOT is_printing*)  THEN 
		uv_power:=0;
		curing_stopped:=TRUE;
		step:=30; 
	END_IF
100://error
	state:=UVLedStateEnum.error;
	error:=TRUE;
	uv_power:=0;
	step:=0; 
	IF SetOff THEN	
		SetOff:=FALSE; 
		step :=200;
	END_IF
200://seting_off		
	SetOff:=FALSE; 
	state:=UVLedStateEnum.setting_off;
	error_code:=UVLedErrorEnum.no_error;
	uv_power:=0;
	off:=TRUE;
	state:=UVLedStateEnum.off;
	step:=0;
END_CASE
IF SetOff OR GVL.Reset THEN 
	step:=200;
END_IF

(*****************ERROR**************************************)
IF 	state<>UVLedStateEnum.setting_off AND state<>UVLedStateEnum.off AND state<>UVLedStateEnum.error THEN 
	error_trig1(CLK:=UVError AND state<>UVLedStateEnum.off , Q=> );
	error_trig2(CLK:=IO_Error AND state<>UVLedStateEnum.off , Q=> );
	IF GVL.Emstop_SAFE THEN 
		error_code:=UVLedErrorEnum.emergency_error;
		step:=100;
	ELSIF error_trig1.Q THEN 
		error_code:=UVLedErrorEnum.abnormal_temperature;
		step:=100;
	ELSIF error_trig2.Q THEN 
		error_code:=UVLedErrorEnum.unknown_error;
		step:=100;
	END_IF
END_IF

	(*******只要速度低于值，就不开灯*****)
IF ABS( Axis[FastScan].Ref.NcToPlc.ActVelo)<=10 THEN
	uv_power:=0;	
END_IF

END_FUNCTION_BLOCK

// ---- POUs/100_SubTank/P_SubTank.TcPOU
PROGRAM P_SubTank
VAR
	FB_SubTankFill_C   :ARRAY[1..12] OF FB_SubTank_C;
	FB_SubTankFill_P   :ARRAY[1..2] OF FB_SubTank_C;
	FB_SubTankFill_W   :ARRAY[1..2] OF FB_SubTank_W;
	FB_SubTankFill_F   :ARRAY[1..2] OF FB_SubTank_W;
	
	PumpWorking1_W,PumpWorking2_W:BOOL;
	PumpWorking1_F,PumpWorking2_F:BOOL;
	
	bqFillPumpWorking_W_r_trig:Tc2_Standard.R_TRIG;//白墨泵启动
	bqFillPumpWorking_F_r_trig:Tc2_Standard.R_TRIG;	//	清洗液泵启动
	
	i:INT;
(****************白墨循坏*******************************)
	FB_Circulation:FB_Circulation;
	
	enable_W_rtrig:Tc2_Standard.R_TRIG;
	enable_F_rtrig:Tc2_Standard.R_TRIG;
END_VAR

VAR PERSISTENT
	SubTankFill_en:ARRAY[1..4] OF BOOL:=[1,1,0,0];//w1,w2,f1,f2  白，清洗液供墨使能
END_VAR

ACT_Color();
ACT_W_F();
ACT_Circulation();
(****white pump**************************************)
stOutput.bqFillPumpWorking[13]:=(PumpWorking1_W ) 
						AND NOT stOutput.bqFillPumpWorking[19] ;
stOutput.bqFillPumpWorking[15]:=(PumpWorking2_W ) 
						AND NOT stOutput.bqFillPumpWorking[20];
(****flush pump**************************************)
stOutput.bqFillPumpWorking[19]:=(PumpWorking1_F ) 
						AND NOT stOutput.bqFillPumpWorking[13] ;
stOutput.bqFillPumpWorking[20]:=(PumpWorking2_F ) 
						AND NOT stOutput.bqFillPumpWorking[15] ;
													
(**********************墨盒里 
		0” circuit not filled (default setting)
	“1” circuit filled with “white ink”
	“2” circuit filled with “storage fluid”
******************************************************)
bqFillPumpWorking_W_r_trig(CLK:=stOutput.bqFillPumpWorking[13] OR stOutput.bqFillPumpWorking[15] , Q=> );
bqFillPumpWorking_F_r_trig(CLK:=stOutput.bqFillPumpWorking[19] OR stOutput.bqFillPumpWorking[20] , Q=> );
IF bqFillPumpWorking_W_r_trig.Q THEN
	SubTankInk_type:=1; 
ELSIF bqFillPumpWorking_F_r_trig.Q THEN 
	SubTankInk_type:=2;
END_IF


(***************切换墨水**************************)
enable_F_rtrig(CLK:= GVL_API.stMU.state=MUStateEnum.swapping AND GVL_API.stMU.cycle=0 , Q=> );
enable_W_rtrig(CLK:=GVL_API.stMU.state=MUStateEnum.swapping AND GVL_API.stMU.cycle=1 , Q=> );
IF enable_W_rtrig.Q THEN  //WHITE
	SubTankFill_en[1]:=TRUE;
	SubTankFill_en[2]:=TRUE;
	SubTankFill_en[3]:=FALSE;
	SubTankFill_en[4]:=FALSE;
ELSIF enable_F_rtrig.Q THEN //FLUSH
	SubTankFill_en[1]:=FALSE;
	SubTankFill_en[2]:=FALSE;
	SubTankFill_en[3]:=TRUE;
	SubTankFill_en[4]:=TRUE;
END_IF

ACTION ACT_Circulation:
FB_Circulation(
	BottomLevel1:=GVL.inklevel_W_L_BOT , 
	BottomLevel2:=GVL.inklevel_W_R_BOT , 
	MUstate:=GVL_API.stMU.state , 
	setoff:= GVL_API.stMU.SetOff OR GVL.Reset, 
	set_pump_voltage1:=HMI_CircPump1_V , 
	set_pump_voltage2:=HMI_CircPump2_V , 
	CircPumpWorking1=>stOutput.bqSubCircPumpWorking[1]  , 
	CircPumpWorking2=> stOutput.bqSubCircPumpWorking[2] , 
	error_code=> ,
	out_pump_voltage1=>EL4002_S[1] , 
	out_pump_voltage2=>EL4002_S[2] );
END_ACTION

ACTION ACT_Color:
(*******************COLOR***************************)
(*
1	:	LC1		2	:	LC2
3	:	LM1		4	:	LM2
5	:	Y1		6	:	Y2
7	:	M1		8	:	M2
9	:	C1		10	:	C2
11	:	K1		12	:	K2
13		P1		14		P2
15		W_L		16		W_R

*)
FOR i:=1 TO 12 DO 
	FB_SubTankFill_C[i](
		sublevel:= stInput.biSubInkTankLevel[i], 
		protectLevel:= stInput.biProtectAirTankLevel_C, 
		filterTime_ON:= T#0S, 
		filterTime_OFF:= T#3S, 
		inkFillTimeOutSet:= inkFillTimeOutSet, 
		PumpWorking=> stOutput.bqFillPumpWorking[i], 
		state=> GVL_API.stSubTank[i].state, 
		error_code=> GVL_API.stSubTank[i].error_code, 
		Error=> GVL_API.stSubTank[i].Error, 
		setoff:=GVL_API.stSubTank[i].Setoff );
END_FOR

(*******************Primer***************************)
	FB_SubTankFill_P[1](
		sublevel:= stInput.biSubInkTankLevel[17], 
		protectLevel:= stInput.biProtectAirTankLevel_W, 
		filterTime_ON:= T#0S, 
		filterTime_OFF:= T#3S, 
		inkFillTimeOutSet:= inkFillTimeOutSet, 
		PumpWorking=> stOutput.bqFillPumpWorking[17], 
		state=> GVL_API.stSubTank[13].state, 
		error_code=> GVL_API.stSubTank[13].error_code, 
		Error=> GVL_API.stSubTank[13].Error, 
		setoff:=GVL_API.stSubTank[13].Setoff );
	FB_SubTankFill_P[2](
		sublevel:= stInput.biSubInkTankLevel[18], 
		protectLevel:= stInput.biProtectAirTankLevel_W, 
		filterTime_ON:= T#0S, 
		filterTime_OFF:= T#3S, 
		inkFillTimeOutSet:= inkFillTimeOutSet, 
		PumpWorking=> stOutput.bqFillPumpWorking[18], 
		state=> GVL_API.stSubTank[14].state, 
		error_code=> GVL_API.stSubTank[14].error_code, 
		Error=> GVL_API.stSubTank[14].Error, 
		setoff:=GVL_API.stSubTank[14].Setoff );
END_ACTION

ACTION ACT_W_F:
(*******************WHITE/FLUSH***************************)	
GVL.inklevel_W_L_BOT:=stInput.biSubInkTankLevel[13] ;	//W_L_BOT
GVL.inklevel_W_L_TOP:=stInput.biSubInkTankLevel[14] ;	//W_L_TOP
GVL.inklevel_W_R_TOP:=stInput.biSubInkTankLevel[15] ;	//W_R_TOP
GVL.inklevel_W_R_BOT:=stInput.biSubInkTankLevel[16] ;	//W_R_BOT


(*******************white***************************)
	FB_SubTankFill_W[1](
		enable:=SubTankFill_en[1],
		fill_in_swap_enable:=GVL.fill_W_in_swap_enable , 
		ISswappingState:=GVL_API.stMU.state  , 
		alternate_fill:= P_MaintenanceUnit.FB_Auto_Cycles_Swap.alternate_Pumping, 
		Toplevel:= GVL.inklevel_W_L_TOP, 
		protectLevel:= stInput.biProtectAirTankLevel_W, 
		filterTime_ON:= T#0S, 
		filterTime_OFF:= T#3S, 
		inkFillTimeOutSet:= inkFillTimeOutSet, 
		CircPumpWorking:= stOutput.bqSubCircPumpWorking[1], 
		PumpWorking=> PumpWorking1_W, 
		state=> GVL_API.stSubTank[15].state, 
		error_code=> GVL_API.stSubTank[15].error_code, 
		Error=> GVL_API.stSubTank[15].Error, 
		setoff:= GVL_API.stSubTank[15].Setoff);
	FB_SubTankFill_W[2](
		enable:=SubTankFill_en[2],
		fill_in_swap_enable:=GVL.fill_W_in_swap_enable , 
		ISswappingState:=GVL_API.stMU.state  , 
		alternate_fill:= P_MaintenanceUnit.FB_Auto_Cycles_Swap.alternate_Pumping, 
		Toplevel:= GVL.inkLevel_W_R_TOP, 
		protectLevel:= stInput.biProtectAirTankLevel_W, 
		filterTime_ON:= T#0S, 
		filterTime_OFF:= T#3S, 
		inkFillTimeOutSet:= inkFillTimeOutSet, 
		CircPumpWorking:= stOutput.bqSubCircPumpWorking[2], 
		PumpWorking=> PumpWorking2_W, 
		state=> GVL_API.stSubTank[16].state, 
		error_code=> GVL_API.stSubTank[16].error_code, 
		Error=> GVL_API.stSubTank[16].Error, 
		setoff:= GVL_API.stSubTank[16].Setoff);	
		
(*******************FLUSH***************************)
	FB_SubTankFill_F[1](
		enable:=SubTankFill_en[3],
		fill_in_swap_enable:=GVL.fill_F_in_swap_enable , 
		ISswappingState:=GVL_API.stMU.state  , 
		alternate_fill:= P_MaintenanceUnit.FB_Auto_Cycles_Swap.alternate_Pumping, 
		Toplevel:= GVL.inklevel_W_L_TOP, 
		protectLevel:= stInput.biProtectAirTankLevel_W, 
		filterTime_ON:= T#0S, 
		filterTime_OFF:= T#3S, 
		inkFillTimeOutSet:= inkFillTimeOutSet, 
		CircPumpWorking:= stOutput.bqSubCircPumpWorking[1], 
		PumpWorking=> PumpWorking1_F, 
		state=> GVL_API.stSubTank[15].state, 
		error_code=> GVL_API.stSubTank[15].error_code, 
		Error=> GVL_API.stSubTank[15].Error, 
		setoff:= GVL_API.stSubTank[15].Setoff);
	FB_SubTankFill_F[2](
		enable:=SubTankFill_en[4],
		fill_in_swap_enable:=GVL.fill_F_in_swap_enable , 
		ISswappingState:=GVL_API.stMU.state  , 
		alternate_fill:= P_MaintenanceUnit.FB_Auto_Cycles_Swap.alternate_Pumping, 
		Toplevel:= GVL.inkLevel_W_R_TOP, 
		protectLevel:= stInput.biProtectAirTankLevel_W, 
		filterTime_ON:= T#0S, 
		filterTime_OFF:= T#3S, 
		inkFillTimeOutSet:= inkFillTimeOutSet, 
		CircPumpWorking:= stOutput.bqSubCircPumpWorking[2], 
		PumpWorking=> PumpWorking2_F, 
		state=> GVL_API.stSubTank[16].state, 
		error_code=> GVL_API.stSubTank[16].error_code, 
		Error=> GVL_API.stSubTank[16].Error, 
		setoff:= GVL_API.stSubTank[16].Setoff);
END_ACTION

END_PROGRAM

// ---- POUs/090MaintenanceUnit/P_MaintenanceUnit.TcPOU
(*换墨  泵输出，通过P_ISS 来控制*)
PROGRAM P_MaintenanceUnit
VAR
	FB_Auto_Cycles_Swap:FB_Auto_Cycles_Swap;//Swap from Ink to Storage Flush
	FB_drip_purge:FB_drip_purge;
	
	log_ErrorEnum:MUErrorEnum;
	log_ID:INT;
	
	log_swapEnum:SwapInfoEnum;
	old_swap_info:INT;
	info_change_ton:Tc2_Standard.TON;
	
	old_dripping_allowed:BOOL;
	ton_dripping_allowed:Tc2_Standard.TON;

END_VAR

ACT_LOG();

(*****************MaintenanceUnit ***************************)
FB_Auto_Cycles_Swap(
	Sensor1:=GVL.inklevel_W_L_TOP  , 
	Sensor4:= GVL.inklevel_W_R_TOP, 
	Circ_Pump_L:= stOutput.bqSubCircPumpWorking[1], 
	Circ_Pump_R:= stOutput.bqSubCircPumpWorking[2], 
	Circ_normal_error:= P_SubTank.FB_Circulation.error_code, 
	btPurge:= stInput.btPurge, 
	state=> GVL_API.stMU.state , 
	error_code=> GVL_API.stMU.error_code, 	
	SwapInfo=>GVL_API.stMU.SwapInfo , 
	VacValve_V8=> , 
	PurValve_V7=> , 
	alternate_Pumping=> , 
	Swapping_Done=> GVL_API.stMU.Swapping_Done, 
	Error=> GVL_API.stMU.Error, 
	initialize:= GVL_API.stMU.Initialize, 
	swap:= GVL_API.stMU.Swap, 
	CYCLE:=GVL_API.stMU.cycle , 
	setoff:=GVL_API.stMU.SetOff );

(**********************三个电磁阀
在自动换墨时，三个电磁阀不受按钮控制********************************)

IF GVL_API.stMU.state=MUStateEnum.swapping THEN 
	stOutput.bqVacValve_W		:=FB_Auto_Cycles_Swap.VacValve_V8;
	stOutput.bqPurValve			:=FB_Auto_Cycles_Swap.PurValve_V7 ;
ELSE
	stOutput.bqVacValve_W		:=stInput.btVacBt_W OR  FB_drip_purge.VacWhiteValve8;
	stOutput.bqVacValve_C		:=stInput.btVacBt_C  OR  FB_drip_purge.VacColorValve9; 
	stOutput.bqPurValve			:=stInput.btPurge     OR  FB_drip_purge.PurgeValve7;
END_IF

(**********************废液位********************************)
IF GVL.MainTankLevel[10]>=3 THEN 
	GVL_API.stMU.waste_maximum_level:=TRUE;
ELSE
	GVL_API.stMU.waste_maximum_level:=FALSE;
END_IF

(**********************FB_drip_purge********************************)
	IntervalTime_W 			:=GVL_API.stMU.IntervalTime_W;
	DripTime_W 				:=GVL_API.stMU.DripTime_W;
	PurgeTime_W 			:=GVL_API.stMU.PurgeTime_W;
	IntervalTime_C 			:=GVL_API.stMU.IntervalTime_C;
	DripTime_C 				:=GVL_API.stMU.DripTime_C;
	PurgeTime_C 			:=GVL_API.stMU.PurgeTime_C ;
FB_drip_purge(
	start_exe:=GVL_API.stMU.dripping_allowed AND GVL_API.stMU.state<>MUStateEnum.swapping  , 
	IntervalTime_W:=IntervalTime_W , 
	DripTime_W:=DripTime_W , 
	PurgeTime_W:=PurgeTime_W , 
	IntervalTime_C:=IntervalTime_C , 
	DripTime_C:=DripTime_C , 
	PurgeTime_C:=PurgeTime_C , 
	PurgeValve7=> , 
	VacWhiteValve8=> , 
	VacColorValve9=> , 
	has_dripped:= GVL_API.stMU.has_dripped);
	

GVL_API.stMU.white_circuit_content:=SubTankInk_type;

ACTION ACT_LOG:
(*************************LOG*******************************************)
log_ID:=550;
//initialize
AlarmActionArray[log_ID+1].AlarmMsg.EN	:=	'MaintenanceUnit  Initialize ';
fbSetAlarm[log_ID+1](
	InUse:=TRUE , 
	EventId:=log_ID+1 , 
	EventActive:=GVL_API.stMU.Initialize , 
	EventClass:=Alm_EventClass.Event , 
	ToTheLogFile:=TRUE, 
	ToTheHistory:=TRUE , 
 );
 //SWAP
 IF GVL_API.stMU.cycle=0 THEN 
	AlarmActionArray[log_ID+2].AlarmMsg.EN	:=	'MaintenanceUnit  Swap Cycle A: Swap white ink to storage ';
ELSIF GVL_API.stMU.cycle=1 THEN 
	AlarmActionArray[log_ID+2].AlarmMsg.EN	:=	'MaintenanceUnit  Swap Cycle B: Swap storage to white ink ';
END_IF

fbSetAlarm[log_ID+2](
	InUse:=TRUE , 
	EventId:=log_ID+2 , 
	EventActive:=GVL_API.stMU.Swap , 
	EventClass:=Alm_EventClass.Event , 
	ToTheLogFile:=TRUE, 
	ToTheHistory:=TRUE , 
 );
 
//ERROR,log_ErrorEnum只能等于一个常数
CASE GVL_API.stMU.error_code OF
0	:	log_ErrorEnum	:=	0	;
1	:	log_ErrorEnum	:=	1	;
2	:	log_ErrorEnum	:=	2	;
3	:	log_ErrorEnum	:=	3	;
4	:	log_ErrorEnum	:=	4	;
5	:	log_ErrorEnum	:=	5	;
6	:	log_ErrorEnum	:=	6	;
7	:	log_ErrorEnum	:=	7	;
8	:	log_ErrorEnum	:=	8	;
9	:	log_ErrorEnum	:=	9	;
666	:	log_ErrorEnum	:=	666	;
END_CASE

AlarmActionArray[log_ID+3].AlarmMsg.EN	:=CONCAT('MaintenanceUnit Error: ',TO_STRING(log_ErrorEnum));
fbSetAlarm[log_ID+3](
	InUse:=TRUE , 
	EventId:=log_ID+3 , 
	EventActive:=GVL_API.stMU.error_code<>0 AND GVL_API.stMU.error_code<>666, 
	EventClass:=Alm_EventClass.Alarm , 
	ToTheLogFile:=TRUE, 
	ToTheHistory:=TRUE , 
 );
 
//reset
AlarmActionArray[log_ID+4].AlarmMsg.EN	:=	'MaintenanceUnit SetOff ';
fbSetAlarm[log_ID+4](
	InUse:=TRUE , 
	EventId:=log_ID+4 , 
	EventActive:=GVL_API.stMU.SetOff , 
	EventClass:=Alm_EventClass.Event , 
	ToTheLogFile:=TRUE, 
	ToTheHistory:=TRUE , 
 );
 
 //dripping_allowed
 IF GVL_API.stMU.dripping_allowed THEN 
 AlarmActionArray[log_ID+5].AlarmMsg.EN	:=	'MaintenanceUnit DrippingAllowed ';
 ELSE
AlarmActionArray[log_ID+5].AlarmMsg.EN	:=	'MaintenanceUnit  Dripping not Allowed ';	 
 END_IF
 
 ton_dripping_allowed(IN:=NOT ton_dripping_allowed.Q  , PT:=T#200MS , Q=> , ET=> );
IF ton_dripping_allowed.Q THEN 
	old_dripping_allowed:= GVL_API.stMU.dripping_allowed  ;
END_IF
 
fbSetAlarm[log_ID+5](
	InUse:=TRUE , 
	EventId:=log_ID+5 , 
	EventActive:=old_dripping_allowed<>GVL_API.stMU.dripping_allowed  , 
	EventClass:=Alm_EventClass.Event , 
	ToTheLogFile:=TRUE, 
	ToTheHistory:=TRUE , 
 );
 
 //has_dripped
  AlarmActionArray[log_ID+6].AlarmMsg.EN	:=	'MaintenanceUnit Has_dripped ';
fbSetAlarm[log_ID+6](
	InUse:=TRUE , 
	EventId:=log_ID+6 , 
	EventActive:=GVL_API.stMU.has_dripped , 
	EventClass:=Alm_EventClass.Event , 
	ToTheLogFile:=TRUE, 
	ToTheHistory:=TRUE , 
 );
  //废液位
  AlarmActionArray[log_ID+7].AlarmMsg.EN	:=	'The maximum level in the waste container is reached ';
fbSetAlarm[log_ID+7](
	InUse:=TRUE , 
	EventId:=log_ID+7 , 
	EventActive:=GVL_API.stMU.waste_maximum_level, 
	EventClass:=Alm_EventClass.Alarm , 
	ToTheLogFile:=TRUE, 
	ToTheHistory:=TRUE , 
 );

 //swap info
 CASE GVL_API.stMU.SwapInfo OF
0	:	log_swapEnum	:=	0	;
1	:	log_swapEnum	:=	1	;
2	:	log_swapEnum	:=	2	;
3	:	log_swapEnum	:=	3	;
4	:	log_swapEnum	:=	4	;
5	:	log_swapEnum	:=	5	;
6	:	log_swapEnum	:=	6	;
7	:	log_swapEnum	:=	7	;
END_CASE
info_change_ton(IN:=NOT info_change_ton.Q  , PT:=T#200MS , Q=> , ET=> );
IF info_change_ton.Q THEN 
	old_swap_info:=GVL_API.stMU.SwapInfo;
END_IF

AlarmActionArray[log_ID+9].AlarmMsg.EN	:=CONCAT('MaintenanceUnit Message: ',TO_STRING(log_swapEnum));
fbSetAlarm[log_ID+9](
	InUse:=TRUE , 
	EventId:=log_ID+9 , 
	EventActive:=old_swap_info<> GVL_API.stMU.SwapInfo, 
	EventClass:=Alm_EventClass.Message , 
	ToTheLogFile:=TRUE, 
	ToTheHistory:=TRUE , 
 );
END_ACTION

END_PROGRAM

// ---- POUs/090MaintenanceUnit/FB/FB_Auto_Cycles_Swap.TcPOU
(**********************SISSI:Swap from Ink to Storage Flush*********************************)
FUNCTION_BLOCK FB_Auto_Cycles_Swap
VAR_INPUT
	Sensor1			:BOOL;
	Sensor4			:BOOL;
	Circ_Pump_L	:BOOL;
	Circ_Pump_R	:BOOL;
	Circ_normal_error:INT;
	btPurge			:BOOL;
	
END_VAR
VAR_OUTPUT
	state								:INT;
	error_code					:INT;
	
